LIN {X 0,Y 336.277,Z 972.972,A -85,B 0,C 180,E1 15001.794,E2 15001.794} C_VEL
LIN {X 0,Y 339.989,Z 961.244,A -85,B 0,C 180,E1 14998.442,E2 14998.442} C_VEL
LIN {X 0,Y 344.835,Z 946.848,A -85,B 0,C 180,E1 14994.971,E2 14994.971} C_VEL
LIN {X 0,Y 349.727,Z 932.706,A -85,B 0,C 180,E1 14992.08,E2 14992.08} C_VEL
LIN {X 0,Y 355.343,Z 916.384,A -85,B 0,C 180,E1 14989.256,E2 14989.256} C_VEL
LIN {X 0,Y 361.12,Z 899.297,A -85,B 0,C 180,E1 14986.734,E2 14986.734} C_VEL
LIN {X 0,Y 367.118,Z 880.482,A -85,B 0,C 180,E1 14984.422,E2 14984.422} C_VEL
LIN {X 0,Y 372.928,Z 861.29,A -85,B 0,C 180,E1 14982.427,E2 14982.427} C_VEL
LIN {X 0,Y 378.209,Z 842.054,A -85,B 0,C 180,E1 14980.766,E2 14980.766} C_VEL
LIN {X 0,Y 383.447,Z 821.063,A -85,B 0,C 180,E1 14979.255,E2 14979.255} C_VEL
LIN {X 0,Y 387.615,Z 801.784,A -85,B 0,C 180,E1 14978.127,E2 14978.127} C_VEL
LIN {X 0,Y 391.771,Z 779.558,A -85,B 0,C 180,E1 14977.076,E2 14977.076} C_VEL
LIN {X 0,Y 394.918,Z 758.505,A -85,B 0,C 180,E1 14976.32,E2 14976.32} C_VEL
LIN {X 0,Y 397.568,Z 734.492,A -85,B 0,C 180,E1 14975.675,E2 14975.675} C_VEL
LIN {X 0,Y 409.561,Z 529.671,A -85,B 0,C 180,E1 14971.616,E2 14971.616} C_VEL
LIN {X 0,Y 411.578,Z 493.902,A -85,B 0,C 180,E1 14970.88,E2 14970.88} C_VEL
LIN {X 0,Y 401.708,Z 478.08,A -85,B 0,C 180,E1 14968.102,E2 14968.102} C_VEL
LIN {X 0,Y 391.949,Z 463.545,A -85,B 0,C 180,E1 14965.053,E2 14965.053} C_VEL
LIN {X 0,Y 383.204,Z 451.285,A -85,B 0,C 180,E1 14961.988,E2 14961.988} C_VEL
LIN {X 0,Y 378.782,Z 445.758,A -85,B 0,C 180,E1 14960.31,E2 14960.31} C_VEL
LIN {X 0,Y 374.764,Z 440.732,A -85,B 0,C 180,E1 14958.672,E2 14958.672} C_VEL
LIN {X 0,Y 370.956,Z 435.952,A -85,B 0,C 180,E1 14957.004,E2 14957.004} C_VEL
LIN {X 0,Y 366.54,Z 430.926,A -85,B 0,C 180,E1 14954.938,E2 14954.938} C_VEL
LIN {X 0,Y 365.222,Z 429.224,A -85,B 0,C 180,E1 14954.263,E2 14954.263} C_VEL
LIN {X 0,Y 361.737,Z 425.607,A -85,B 0,C 180,E1 14952.45,E2 14952.45} C_VEL
LIN {X 0,Y 360.146,Z 423.216,A -85,B 0,C 180,E1 14951.508,E2 14951.508} C_VEL
LIN {X 0,Y 356.524,Z 419.861,A -85,B 0,C 180,E1 14949.361,E2 14949.361} C_VEL
LIN {X 0,Y 354.747,Z 416.927,A -85,B 0,C 180,E1 14948.101,E2 14948.101} C_VEL
LIN {X 0,Y 351.223,Z 414.2,A -85,B 0,C 180,E1 14945.636,E2 14945.636} C_VEL
LIN {X 0,Y 349.164,Z 410.557,A -85,B 0,C 180,E1 14943.776,E2 14943.776} C_VEL
LIN {X 0,Y 345.15,Z 407.759,A -85,B 0,C 180,E1 14939.999,E2 14939.999} C_VEL
LIN {X 0,Y 342.976,Z 403.947,A -85,B 0,C 180,E1 14936.991,E2 14936.991} C_VEL
LIN {X 0,Y 339.469,Z 401.855,A -85,B 0,C 180,E1 14929.992,E2 14929.992} C_VEL
LIN {X 0,Y 338.898,Z 401.219,A -85,B 0,C 180,E1 14924.715,E2 14924.715} C_VEL
LIN {X 0,Y 340.368,Z 402.502,A -85,B 0,C 180,E1 14918.605,E2 14918.605} C_VEL
LIN {X 0,Y 343.058,Z 404.045,A -85,B 0,C 180,E1 14914.075,E2 14914.075} C_VEL
LIN {X 0,Y 345.939,Z 408.538,A -85,B 0,C 180,E1 14910.38,E2 14910.38} C_VEL
LIN {X 0,Y 349.443,Z 410.923,A -85,B 0,C 180,E1 14907.213,E2 14907.213} C_VEL
LIN {X 0,Y 351.487,Z 414.448,A -85,B 0,C 180,E1 14905.423,E2 14905.423} C_VEL
LIN {X 0,Y 355.199,Z 417.46,A -85,B 0,C 180,E1 14902.857,E2 14902.857} C_VEL
LIN {X 0,Y 357.603,Z 421.145,A -85,B 0,C 180,E1 14901.221,E2 14901.221} C_VEL
LIN {X 0,Y 360.71,Z 423.864,A -85,B 0,C 180,E1 14899.446,E2 14899.446} C_VEL
LIN {X 0,Y 363.718,Z 427.939,A -85,B 0,C 180,E1 14897.768,E2 14897.768} C_VEL
LIN {X 0,Y 365.997,Z 430.022,A -85,B 0,C 180,E1 14896.637,E2 14896.637} C_VEL
LIN {X 0,Y 369.557,Z 434.555,A -85,B 0,C 180,E1 14894.914,E2 14894.914} C_VEL
LIN {X 0,Y 371.282,Z 436.471,A -85,B 0,C 180,E1 14894.136,E2 14894.136} C_VEL
LIN {X 0,Y 375.26,Z 441.146,A -85,B 0,C 180,E1 14892.433,E2 14892.433} C_VEL
LIN {X 0,Y 379.777,Z 446.735,A -85,B 0,C 180,E1 14890.627,E2 14890.627} C_VEL
LIN {X 0,Y 388.837,Z 458.356,A -85,B 0,C 180,E1 14887.355,E2 14887.355} C_VEL
LIN {X 0,Y 399.329,Z 472.434,A -85,B 0,C 180,E1 14884.026,E2 14884.026} C_VEL
LIN {X 0,Y 409.84,Z 487.637,A -85,B 0,C 180,E1 14881.057,E2 14881.057} C_VEL
LIN {X 0,Y 411.391,Z 490.242,A -85,B 0,C 180,E1 14880.637,E2 14880.637} C_VEL
LIN {X 0,Y 399.236,Z 697.815,A -85,B 0,C 180,E1 14876.553,E2 14876.553} C_VEL
LIN {X 0,Y 397.171,Z 724.706,A -85,B 0,C 180,E1 14875.953,E2 14875.953} C_VEL
LIN {X 0,Y 394.429,Z 747.684,A -85,B 0,C 180,E1 14875.24,E2 14875.24} C_VEL
LIN {X 0,Y 390.892,Z 769.549,A -85,B 0,C 180,E1 14874.313,E2 14874.313} C_VEL
LIN {X 0,Y 386.65,Z 791.514,A -85,B 0,C 180,E1 14873.139,E2 14873.139} C_VEL
LIN {X 0,Y 382.044,Z 811.473,A -85,B 0,C 180,E1 14871.81,E2 14871.81} C_VEL
LIN {X 0,Y 376.547,Z 832.601,A -85,B 0,C 180,E1 14870.107,E2 14870.107} C_VEL
LIN {X 0,Y 371.312,Z 850.638,A -85,B 0,C 180,E1 14868.358,E2 14868.358} C_VEL
LIN {X 0,Y 365.02,Z 870.569,A -85,B 0,C 180,E1 14866.055,E2 14866.055} C_VEL
LIN {X 0,Y 359.424,Z 887.312,A -85,B 0,C 180,E1 14863.754,E2 14863.754} C_VEL
LIN {X 0,Y 353.658,Z 903.672,A -85,B 0,C 180,E1 14861.079,E2 14861.079} C_VEL
LIN {X 0,Y 348.373,Z 918.498,A -85,B 0,C 180,E1 14858.245,E2 14858.245} C_VEL
LIN {X 0,Y 345.359,Z 926.835,A -85,B 0,C 180,E1 14856.41,E2 14856.41} C_VEL
LIN {X 0,Y 342.903,Z 931.412,A -85,B 0,C 180,E1 14855.448,E2 14855.448} C_VEL
LIN {X 0,Y 333.624,Z 942.542,A -85,B 0,C 180,E1 14853.077,E2 14853.077} C_VEL
LIN {X 0,Y 331.307,Z 946.444,A -85,B 0,C 180,E1 14851.991,E2 14851.991} C_VEL
LIN {X 0,Y 327.771,Z 956.623,A -85,B 0,C 180,E1 14848.596,E2 14848.596} C_VEL
LIN {X 0,Y 324.573,Z 966.727,A -85,B 0,C 180,E1 14844.515,E2 14844.515} C_VEL
LIN {X 0,Y 322.438,Z 974.749,A -85,B 0,C 180,E1 14840.535,E2 14840.535} C_VEL
LIN {X 0,Y 321.058,Z 981.036,A -85,B 0,C 180,E1 14836.488,E2 14836.488} C_VEL
LIN {X 0,Y 320.354,Z 985.736,A -85,B 0,C 180,E1 14832.56,E2 14832.56} C_VEL
LIN {X 0,Y 320.061,Z 988.751,A -85,B 0,C 180,E1 14828.749,E2 14828.749} C_VEL
LIN {X 0,Y 319.978,Z 990.434,A -85,B 0,C 180,E1 14825.241,E2 14825.241} C_VEL
LIN {X 0,Y 319.967,Z 990.942,A -85,B 0,C 180,E1 14821.229,E2 14821.229} C_VEL
LIN {X 0,Y 319.978,Z 990.216,A -85,B 0,C 180,E1 14817.868,E2 14817.868} C_VEL
LIN {X 0,Y 320.126,Z 988.191,A -85,B 0,C 180,E1 14813.994,E2 14813.994} C_VEL
LIN {X 0,Y 320.55,Z 984.512,A -85,B 0,C 180,E1 14810.012,E2 14810.012} C_VEL
LIN {X 0,Y 321.476,Z 979.566,A -85,B 0,C 180,E1 14806.081,E2 14806.081} C_VEL
LIN {X 0,Y 323.018,Z 973.025,A -85,B 0,C 180,E1 14802.199,E2 14802.199} C_VEL
LIN {X 0,Y 325.366,Z 965.15,A -85,B 0,C 180,E1 14798.372,E2 14798.372} C_VEL
LIN {X 0,Y 328.589,Z 955.458,A -85,B 0,C 180,E1 14794.59,E2 14794.59} C_VEL
LIN {X 0,Y 332.897,Z 943.804,A -85,B 0,C 180,E1 14790.789,E2 14790.789} C_VEL
LIN {X 0,Y 337.523,Z 931.777,A -85,B 0,C 180,E1 14787.525,E2 14787.525} C_VEL
LIN {X 0,Y 343.347,Z 917.072,A -85,B 0,C 180,E1 14784.169,E2 14784.169} C_VEL
LIN {X 0,Y 349.136,Z 902.312,A -85,B 0,C 180,E1 14781.329,E2 14781.329} C_VEL
LIN {X 0,Y 355.55,Z 885.443,A -85,B 0,C 180,E1 14778.605,E2 14778.605} C_VEL
LIN {X 0,Y 362.016,Z 867.798,A -85,B 0,C 180,E1 14776.198,E2 14776.198} C_VEL
LIN {X 0,Y 368.118,Z 849.666,A -85,B 0,C 180,E1 14774.139,E2 14774.139} C_VEL
LIN {X 0,Y 374.231,Z 830.086,A -85,B 0,C 180,E1 14772.264,E2 14772.264} C_VEL
LIN {X 0,Y 379.729,Z 810.272,A -85,B 0,C 180,E1 14770.699,E2 14770.699} C_VEL
LIN {X 0,Y 385.279,Z 787.324,A -85,B 0,C 180,E1 14769.222,E2 14769.222} C_VEL
LIN {X 0,Y 389.546,Z 766.561,A -85,B 0,C 180,E1 14768.153,E2 14768.153} C_VEL
LIN {X 0,Y 393.289,Z 743.628,A -85,B 0,C 180,E1 14767.242,E2 14767.242} C_VEL
LIN {X 0,Y 396.188,Z 720.474,A -85,B 0,C 180,E1 14766.565,E2 14766.565} C_VEL
LIN {X 0,Y 403.462,Z 618.117,A -85,B 0,C 180,E1 14764.456,E2 14764.456} C_VEL
LIN {X 0,Y 412.474,Z 496.118,A -85,B 0,C 180,E1 14761.945,E2 14761.945} C_VEL
LIN {X 0,Y 406.567,Z 486.319,A -85,B 0,C 180,E1 14759.578,E2 14759.578} C_VEL
LIN {X 0,Y 401.968,Z 478.937,A -85,B 0,C 180,E1 14757.363,E2 14757.363} C_VEL
LIN {X 0,Y 399.286,Z 474.781,A -85,B 0,C 180,E1 14755.836,E2 14755.836} C_VEL
LIN {X 0,Y 396.693,Z 470.696,A -85,B 0,C 180,E1 14754.069,E2 14754.069} C_VEL
LIN {X 0,Y 394.074,Z 466.488,A -85,B 0,C 180,E1 14751.685,E2 14751.685} C_VEL
LIN {X 0,Y 393.166,Z 465.528,A -85,B 0,C 180,E1 14750.634,E2 14750.634} C_VEL
LIN {X 0,Y 391.561,Z 463.129,A -85,B 0,C 180,E1 14746.638,E2 14746.638} C_VEL
LIN {X 0,Y 391.761,Z 463.738,A -85,B 0,C 180,E1 14744.456,E2 14744.456} C_VEL
LIN {X 0,Y 394.02,Z 466.346,A -85,B 0,C 180,E1 14740.816,E2 14740.816} C_VEL
LIN {X 0,Y 396.488,Z 470.513,A -85,B 0,C 180,E1 14738.525,E2 14738.525} C_VEL
LIN {X 0,Y 397.564,Z 472.154,A -85,B 0,C 180,E1 14737.729,E2 14737.729} C_VEL
LIN {X 0,Y 400.699,Z 477.067,A -85,B 0,C 180,E1 14735.766,E2 14735.766} C_VEL
LIN {X 0,Y 405.039,Z 484.946,A -85,B 0,C 180,E1 14733.501,E2 14733.501} C_VEL
LIN {X 0,Y 410.015,Z 494.373,A -85,B 0,C 180,E1 14731.329,E2 14731.329} C_VEL
LIN {X 0,Y 412.455,Z 499.516,A -85,B 0,C 180,E1 14730.365,E2 14730.365} C_VEL
LIN {X 0,Y 398.746,Z 689.757,A -85,B 0,C 180,E1 14726.482,E2 14726.482} C_VEL
LIN {X 0,Y 395.345,Z 736.083,A -85,B 0,C 180,E1 14725.504,E2 14725.504} C_VEL
LIN {X 0,Y 392.335,Z 758.929,A -85,B 0,C 180,E1 14724.859,E2 14724.859} C_VEL
LIN {X 0,Y 388.399,Z 781.737,A -85,B 0,C 180,E1 14724,E2 14724} C_VEL
LIN {X 0,Y 384.215,Z 801.576,A -85,B 0,C 180,E1 14723.031,E2 14723.031} C_VEL
LIN {X 0,Y 378.701,Z 824.282,A -85,B 0,C 180,E1 14721.647,E2 14721.647} C_VEL
LIN {X 0,Y 373.434,Z 843.326,A -85,B 0,C 180,E1 14720.218,E2 14720.218} C_VEL
LIN {X 0,Y 366.723,Z 865.269,A -85,B 0,C 180,E1 14718.223,E2 14718.223} C_VEL
LIN {X 0,Y 360.501,Z 884.173,A -85,B 0,C 180,E1 14716.151,E2 14716.151} C_VEL
LIN {X 0,Y 354.121,Z 902.261,A -85,B 0,C 180,E1 14713.774,E2 14713.774} C_VEL
LIN {X 0,Y 347.818,Z 919.74,A -85,B 0,C 180,E1 14711.066,E2 14711.066} C_VEL
LIN {X 0,Y 341.862,Z 935.706,A -85,B 0,C 180,E1 14708.111,E2 14708.111} C_VEL
LIN {X 0,Y 336.071,Z 951.541,A -85,B 0,C 180,E1 14704.633,E2 14704.633} C_VEL
LIN {X 0,Y 331.503,Z 964.51,A -85,B 0,C 180,E1 14701.255,E2 14701.255} C_VEL
LIN {X 0,Y 327.475,Z 976.677,A -85,B 0,C 180,E1 14697.459,E2 14697.459} C_VEL
LIN {X 0,Y 324.466,Z 987.037,A -85,B 0,C 180,E1 14693.621,E2 14693.621} C_VEL
LIN {X 0,Y 322.36,Z 995.464,A -85,B 0,C 180,E1 14689.765,E2 14689.765} C_VEL
LIN {X 0,Y 320.975,Z 1002.68,A -85,B 0,C 180,E1 14685.729,E2 14685.729} C_VEL
LIN {X 0,Y 320.293,Z 1007.657,A -85,B 0,C 180,E1 14682.078,E2 14682.078} C_VEL
LIN {X 0,Y 320.024,Z 1011.558,A -85,B 0,C 180,E1 14678.268,E2 14678.268} C_VEL
LIN {X 0,Y 319.947,Z 1013.919,A -85,B 0,C 180,E1 14674.486,E2 14674.486} C_VEL
LIN {X 0,Y 319.954,Z 1014.85,A -85,B 0,C 180,E1 14671.259,E2 14671.259} C_VEL
LIN {X 0,Y 319.957,Z 1014.756,A -85,B 0,C 180,E1 14667.856,E2 14667.856} C_VEL
LIN {X 0,Y 319.961,Z 1013.15,A -85,B 0,C 180,E1 14663.907,E2 14663.907} C_VEL
LIN {X 0,Y 320.07,Z 1010.516,A -85,B 0,C 180,E1 14660.476,E2 14660.476} C_VEL
LIN {X 0,Y 320.522,Z 1006.051,A -85,B 0,C 180,E1 14656.476,E2 14656.476} C_VEL
LIN {X 0,Y 321.458,Z 1000.137,A -85,B 0,C 180,E1 14652.633,E2 14652.633} C_VEL
LIN {X 0,Y 323.16,Z 992.342,A -85,B 0,C 180,E1 14648.593,E2 14648.593} C_VEL
LIN {X 0,Y 325.507,Z 983.552,A -85,B 0,C 180,E1 14644.926,E2 14644.926} C_VEL
LIN {X 0,Y 328.905,Z 972.591,A -85,B 0,C 180,E1 14641.103,E2 14641.103} C_VEL
LIN {X 0,Y 332.857,Z 960.835,A -85,B 0,C 180,E1 14637.685,E2 14637.685} C_VEL
LIN {X 0,Y 337.971,Z 946.399,A -85,B 0,C 180,E1 14634.151,E2 14634.151} C_VEL
LIN {X 0,Y 343.469,Z 931.373,A -85,B 0,C 180,E1 14631.048,E2 14631.048} C_VEL
LIN {X 0,Y 349.382,Z 914.816,A -85,B 0,C 180,E1 14628.188,E2 14628.188} C_VEL
LIN {X 0,Y 355.647,Z 896.985,A -85,B 0,C 180,E1 14625.579,E2 14625.579} C_VEL
LIN {X 0,Y 361.661,Z 878.859,A -85,B 0,C 180,E1 14623.366,E2 14623.366} C_VEL
LIN {X 0,Y 368.154,Z 857.85,A -85,B 0,C 180,E1 14621.22,E2 14621.22} C_VEL
LIN {X 0,Y 373.6,Z 838.56,A -85,B 0,C 180,E1 14619.587,E2 14619.587} C_VEL
LIN {X 0,Y 378.791,Z 817.787,A -85,B 0,C 180,E1 14618.141,E2 14618.141} C_VEL
LIN {X 0,Y 383.417,Z 796.805,A -85,B 0,C 180,E1 14616.949,E2 14616.949} C_VEL
LIN {X 0,Y 387.543,Z 774.028,A -85,B 0,C 180,E1 14615.94,E2 14615.94} C_VEL
LIN {X 0,Y 390.938,Z 751.015,A -85,B 0,C 180,E1 14615.171,E2 14615.171} C_VEL
LIN {X 0,Y 393.173,Z 727.848,A -85,B 0,C 180,E1 14614.609,E2 14614.609} C_VEL
LIN {X 0,Y 405.857,Z 518.019,A -85,B 0,C 180,E1 14610.446,E2 14610.446} C_VEL
LIN {X 0,Y 407.024,Z 498.197,A -85,B 0,C 180,E1 14610.033,E2 14610.033} C_VEL
LIN {X 0,Y 398.344,Z 484.149,A -85,B 0,C 180,E1 14607.506,E2 14607.506} C_VEL
LIN {X 0,Y 389.062,Z 470.099,A -85,B 0,C 180,E1 14604.521,E2 14604.521} C_VEL
LIN {X 0,Y 380.64,Z 458.182,A -85,B 0,C 180,E1 14601.495,E2 14601.495} C_VEL
LIN {X 0,Y 376.458,Z 452.884,A -85,B 0,C 180,E1 14599.874,E2 14599.874} C_VEL
LIN {X 0,Y 372.491,Z 447.9,A -85,B 0,C 180,E1 14598.222,E2 14598.222} C_VEL
LIN {X 0,Y 368.096,Z 442.463,A -85,B 0,C 180,E1 14596.246,E2 14596.246} C_VEL
LIN {X 0,Y 364.285,Z 437.786,A -85,B 0,C 180,E1 14594.382,E2 14594.382} C_VEL
LIN {X 0,Y 359.675,Z 432.659,A -85,B 0,C 180,E1 14591.93,E2 14591.93} C_VEL
LIN {X 0,Y 358.575,Z 430.922,A -85,B 0,C 180,E1 14591.255,E2 14591.255} C_VEL
LIN {X 0,Y 354.951,Z 427.511,A -85,B 0,C 180,E1 14589.075,E2 14589.075} C_VEL
LIN {X 0,Y 353.175,Z 424.649,A -85,B 0,C 180,E1 14587.801,E2 14587.801} C_VEL
LIN {X 0,Y 349.731,Z 421.837,A -85,B 0,C 180,E1 14585.331,E2 14585.331} C_VEL
LIN {X 0,Y 347.677,Z 418.278,A -85,B 0,C 180,E1 14583.462,E2 14583.462} C_VEL
LIN {X 0,Y 343.903,Z 415.6,A -85,B 0,C 180,E1 14579.833,E2 14579.833} C_VEL
LIN {X 0,Y 341.756,Z 411.788,A -85,B 0,C 180,E1 14576.813,E2 14576.813} C_VEL
LIN {X 0,Y 338.282,Z 409.684,A -85,B 0,C 180,E1 14569.612,E2 14569.612} C_VEL
LIN {X 0,Y 337.832,Z 409.17,A -85,B 0,C 180,E1 14564.551,E2 14564.551} C_VEL
LIN {X 0,Y 339.384,Z 410.502,A -85,B 0,C 180,E1 14558.391,E2 14558.391} C_VEL
LIN {X 0,Y 341.903,Z 411.948,A -85,B 0,C 180,E1 14554.167,E2 14554.167} C_VEL
LIN {X 0,Y 344.433,Z 416.115,A -85,B 0,C 180,E1 14550.81,E2 14550.81} C_VEL
LIN {X 0,Y 347.994,Z 418.665,A -85,B 0,C 180,E1 14547.5,E2 14547.5} C_VEL
LIN {X 0,Y 350.185,Z 422.312,A -85,B 0,C 180,E1 14545.574,E2 14545.574} C_VEL
LIN {X 0,Y 353.601,Z 425.138,A -85,B 0,C 180,E1 14543.168,E2 14543.168} C_VEL
LIN {X 0,Y 356.254,Z 429.032,A -85,B 0,C 180,E1 14541.356,E2 14541.356} C_VEL
LIN {X 0,Y 359.022,Z 431.532,A -85,B 0,C 180,E1 14539.75,E2 14539.75} C_VEL
LIN {X 0,Y 362.254,Z 435.766,A -85,B 0,C 180,E1 14537.932,E2 14537.932} C_VEL
LIN {X 0,Y 364.229,Z 437.693,A -85,B 0,C 180,E1 14536.932,E2 14536.932} C_VEL
LIN {X 0,Y 367.883,Z 442.241,A -85,B 0,C 180,E1 14535.146,E2 14535.146} C_VEL
LIN {X 0,Y 369.66,Z 444.453,A -85,B 0,C 180,E1 14534.321,E2 14534.321} C_VEL
LIN {X 0,Y 374.201,Z 450.014,A -85,B 0,C 180,E1 14532.358,E2 14532.358} C_VEL
LIN {X 0,Y 378.931,Z 455.989,A -85,B 0,C 180,E1 14530.466,E2 14530.466} C_VEL
LIN {X 0,Y 384.137,Z 462.62,A -85,B 0,C 180,E1 14528.54,E2 14528.54} C_VEL
LIN {X 0,Y 391.773,Z 472.822,A -85,B 0,C 180,E1 14525.954,E2 14525.954} C_VEL
LIN {X 0,Y 399.937,Z 484.207,A -85,B 0,C 180,E1 14523.447,E2 14523.447} C_VEL
LIN {X 0,Y 406.789,Z 494.512,A -85,B 0,C 180,E1 14521.499,E2 14521.499} C_VEL
LIN {X 0,Y 394.119,Z 703.148,A -85,B 0,C 180,E1 14517.375,E2 14517.375} C_VEL
LIN {X 0,Y 392.075,Z 726.879,A -85,B 0,C 180,E1 14516.82,E2 14516.82} C_VEL
LIN {X 0,Y 389.066,Z 750.34,A -85,B 0,C 180,E1 14516.063,E2 14516.063} C_VEL
LIN {X 0,Y 385.671,Z 770.502,A -85,B 0,C 180,E1 14515.197,E2 14515.197} C_VEL
LIN {X 0,Y 381.161,Z 792.857,A -85,B 0,C 180,E1 14513.985,E2 14513.985} C_VEL
LIN {X 0,Y 376.645,Z 811.811,A -85,B 0,C 180,E1 14512.715,E2 14512.715} C_VEL
LIN {X 0,Y 370.955,Z 832.98,A -85,B 0,C 180,E1 14511.001,E2 14511.001} C_VEL
LIN {X 0,Y 365.525,Z 851.03,A -85,B 0,C 180,E1 14509.24,E2 14509.24} C_VEL
LIN {X 0,Y 358.981,Z 870.958,A -85,B 0,C 180,E1 14506.916,E2 14506.916} C_VEL
LIN {X 0,Y 352.971,Z 888.244,A -85,B 0,C 180,E1 14504.513,E2 14504.513} C_VEL
LIN {X 0,Y 346.968,Z 904.539,A -85,B 0,C 180,E1 14501.801,E2 14501.801} C_VEL
LIN {X 0,Y 341.454,Z 919.307,A -85,B 0,C 180,E1 14498.923,E2 14498.923} C_VEL
LIN {X 0,Y 336.346,Z 932.716,A -85,B 0,C 180,E1 14495.795,E2 14495.795} C_VEL
LIN {X 0,Y 331.601,Z 945.647,A -85,B 0,C 180,E1 14492.241,E2 14492.241} C_VEL
LIN {X 0,Y 331.307,Z 946.444,A -85,B 0,C 180,E1 14491.991,E2 14491.991} C_VEL
LIN {X 0,Y 329.061,Z 950.294,A -85,B 0,C 180,E1 14490.878,E2 14490.878} C_VEL
LIN {X 0,Y 319.962,Z 960.084,A -85,B 0,C 180,E1 14487.96,E2 14487.96} C_VEL
LIN {X 0,Y 318.317,Z 962.79,A -85,B 0,C 180,E1 14486.915,E2 14486.915} C_VEL
LIN {X 0,Y 315.495,Z 971.833,A -85,B 0,C 180,E1 14482.712,E2 14482.712} C_VEL
LIN {X 0,Y 313.818,Z 978.282,A -85,B 0,C 180,E1 14478.974,E2 14478.974} C_VEL
LIN {X 0,Y 312.664,Z 984.089,A -85,B 0,C 180,E1 14474.603,E2 14474.603} C_VEL
LIN {X 0,Y 312.198,Z 987.465,A -85,B 0,C 180,E1 14471.122,E2 14471.122} C_VEL
LIN {X 0,Y 312.007,Z 990.048,A -85,B 0,C 180,E1 14467.18,E2 14467.18} C_VEL
LIN {X 0,Y 311.956,Z 991.133,A -85,B 0,C 180,E1 14463.411,E2 14463.411} C_VEL
LIN {X 0,Y 311.954,Z 991.112,A -85,B 0,C 180,E1 14459.995,E2 14459.995} C_VEL
LIN {X 0,Y 312.018,Z 989.858,A -85,B 0,C 180,E1 14456.096,E2 14456.096} C_VEL
LIN {X 0,Y 312.24,Z 987.471,A -85,B 0,C 180,E1 14452.519,E2 14452.519} C_VEL
LIN {X 0,Y 312.812,Z 983.758,A -85,B 0,C 180,E1 14448.691,E2 14448.691} C_VEL
LIN {X 0,Y 314.044,Z 978.025,A -85,B 0,C 180,E1 14444.463,E2 14444.463} C_VEL
LIN {X 0,Y 316.104,Z 970.865,A -85,B 0,C 180,E1 14440.327,E2 14440.327} C_VEL
LIN {X 0,Y 319.007,Z 962.036,A -85,B 0,C 180,E1 14436.327,E2 14436.327} C_VEL
LIN {X 0,Y 323.03,Z 951.337,A -85,B 0,C 180,E1 14432.321,E2 14432.321} C_VEL
LIN {X 0,Y 327.537,Z 940.002,A -85,B 0,C 180,E1 14428.816,E2 14428.816} C_VEL
LIN {X 0,Y 333.312,Z 926.039,A -85,B 0,C 180,E1 14425.213,E2 14425.213} C_VEL
LIN {X 0,Y 339.437,Z 911.427,A -85,B 0,C 180,E1 14422.051,E2 14422.051} C_VEL
LIN {X 0,Y 345.741,Z 895.864,A -85,B 0,C 180,E1 14419.25,E2 14419.25} C_VEL
LIN {X 0,Y 352.634,Z 878.365,A -85,B 0,C 180,E1 14416.582,E2 14416.582} C_VEL
LIN {X 0,Y 359.144,Z 860.624,A -85,B 0,C 180,E1 14414.332,E2 14414.332} C_VEL
LIN {X 0,Y 366.174,Z 840,A -85,B 0,C 180,E1 14412.155,E2 14412.155} C_VEL
LIN {X 0,Y 372.151,Z 820.633,A -85,B 0,C 180,E1 14410.462,E2 14410.462} C_VEL
LIN {X 0,Y 377.731,Z 800.016,A -85,B 0,C 180,E1 14408.985,E2 14408.985} C_VEL
LIN {X 0,Y 382.61,Z 779.456,A -85,B 0,C 180,E1 14407.777,E2 14407.777} C_VEL
LIN {X 0,Y 386.801,Z 757.712,A -85,B 0,C 180,E1 14406.771,E2 14406.771} C_VEL
LIN {X 0,Y 390.304,Z 735.408,A -85,B 0,C 180,E1 14405.971,E2 14405.971} C_VEL
LIN {X 0,Y 392.742,Z 712.745,A -85,B 0,C 180,E1 14405.391,E2 14405.391} C_VEL
LIN {X 0,Y 408.409,Z 506.179,A -85,B 0,C 180,E1 14401.154,E2 14401.154} C_VEL
LIN {X 0,Y 408.741,Z 500.898,A -85,B 0,C 180,E1 14401.017,E2 14401.017} C_VEL
LIN {X 0,Y 403.256,Z 491.362,A -85,B 0,C 180,E1 14398.615,E2 14398.615} C_VEL
LIN {X 0,Y 398.357,Z 483.284,A -85,B 0,C 180,E1 14395.971,E2 14395.971} C_VEL
LIN {X 0,Y 395.153,Z 478.287,A -85,B 0,C 180,E1 14393.754,E2 14393.754} C_VEL
LIN {X 0,Y 392.674,Z 474.041,A -85,B 0,C 180,E1 14391.36,E2 14391.36} C_VEL
LIN {X 0,Y 390.494,Z 471.172,A -85,B 0,C 180,E1 14386.979,E2 14386.979} C_VEL
LIN {X 0,Y 390.535,Z 471.273,A -85,B 0,C 180,E1 14385.166,E2 14385.166} C_VEL
LIN {X 0,Y 392.754,Z 474.252,A -85,B 0,C 180,E1 14380.983,E2 14380.983} C_VEL
LIN {X 0,Y 395.22,Z 478.394,A -85,B 0,C 180,E1 14378.636,E2 14378.636} C_VEL
LIN {X 0,Y 398.844,Z 484.355,A -85,B 0,C 180,E1 14376.157,E2 14376.157} C_VEL
LIN {X 0,Y 403.442,Z 492.993,A -85,B 0,C 180,E1 14373.666,E2 14373.666} C_VEL
LIN {X 0,Y 408.76,Z 503.676,A -85,B 0,C 180,E1 14371.298,E2 14371.298} C_VEL
LIN {X 0,Y 394.509,Z 692.288,A -85,B 0,C 180,E1 14367.431,E2 14367.431} C_VEL
LIN {X 0,Y 391.129,Z 736.031,A -85,B 0,C 180,E1 14366.501,E2 14366.501} C_VEL
LIN {X 0,Y 387.99,Z 758.915,A -85,B 0,C 180,E1 14365.852,E2 14365.852} C_VEL
LIN {X 0,Y 383.757,Z 782.304,A -85,B 0,C 180,E1 14364.966,E2 14364.966} C_VEL
LIN {X 0,Y 379.442,Z 801.994,A -85,B 0,C 180,E1 14364,E2 14364} C_VEL
LIN {X 0,Y 373.735,Z 824.467,A -85,B 0,C 180,E1 14362.619,E2 14362.619} C_VEL
LIN {X 0,Y 368.279,Z 843.4,A -85,B 0,C 180,E1 14361.191,E2 14361.191} C_VEL
LIN {X 0,Y 361.533,Z 864.591,A -85,B 0,C 180,E1 14359.257,E2 14359.257} C_VEL
LIN {X 0,Y 355.068,Z 883.393,A -85,B 0,C 180,E1 14357.19,E2 14357.19} C_VEL
LIN {X 0,Y 348.379,Z 901.522,A -85,B 0,C 180,E1 14354.801,E2 14354.801} C_VEL
LIN {X 0,Y 341.762,Z 919.046,A -85,B 0,C 180,E1 14352.069,E2 14352.069} C_VEL
LIN {X 0,Y 335.651,Z 934.584,A -85,B 0,C 180,E1 14349.167,E2 14349.167} C_VEL
LIN {X 0,Y 329.765,Z 949.824,A -85,B 0,C 180,E1 14345.821,E2 14345.821} C_VEL
LIN {X 0,Y 325.024,Z 962.319,A -85,B 0,C 180,E1 14342.554,E2 14342.554} C_VEL
LIN {X 0,Y 320.431,Z 975.307,A -85,B 0,C 180,E1 14338.522,E2 14338.522} C_VEL
LIN {X 0,Y 317.245,Z 985.323,A -85,B 0,C 180,E1 14334.787,E2 14334.787} C_VEL
LIN {X 0,Y 314.754,Z 994.417,A -85,B 0,C 180,E1 14330.652,E2 14330.652} C_VEL
LIN {X 0,Y 313.242,Z 1001.486,A -85,B 0,C 180,E1 14326.7,E2 14326.7} C_VEL
LIN {X 0,Y 312.366,Z 1007.132,A -85,B 0,C 180,E1 14322.577,E2 14322.577} C_VEL
LIN {X 0,Y 312.043,Z 1010.919,A -85,B 0,C 180,E1 14318.853,E2 14318.853} C_VEL
LIN {X 0,Y 311.95,Z 1013.545,A -85,B 0,C 180,E1 14314.786,E2 14314.786} C_VEL
LIN {X 0,Y 311.96,Z 1014.55,A -85,B 0,C 180,E1 14311.291,E2 14311.291} C_VEL
LIN {X 0,Y 311.961,Z 1014.456,A -85,B 0,C 180,E1 14307.801,E2 14307.801} C_VEL
LIN {X 0,Y 311.968,Z 1012.846,A -85,B 0,C 180,E1 14303.75,E2 14303.75} C_VEL
LIN {X 0,Y 312.079,Z 1010.206,A -85,B 0,C 180,E1 14300.23,E2 14300.23} C_VEL
LIN {X 0,Y 312.579,Z 1005.727,A -85,B 0,C 180,E1 14296.125,E2 14296.125} C_VEL
LIN {X 0,Y 313.531,Z 1000.115,A -85,B 0,C 180,E1 14292.371,E2 14292.371} C_VEL
LIN {X 0,Y 315.297,Z 992.563,A -85,B 0,C 180,E1 14288.301,E2 14288.301} C_VEL
LIN {X 0,Y 317.808,Z 983.659,A -85,B 0,C 180,E1 14284.475,E2 14284.475} C_VEL
LIN {X 0,Y 321.388,Z 972.777,A -85,B 0,C 180,E1 14280.565,E2 14280.565} C_VEL
LIN {X 0,Y 325.536,Z 961.068,A -85,B 0,C 180,E1 14277.076,E2 14277.076} C_VEL
LIN {X 0,Y 330.892,Z 946.734,A -85,B 0,C 180,E1 14273.476,E2 14273.476} C_VEL
LIN {X 0,Y 336.28,Z 932.608,A -85,B 0,C 180,E1 14270.493,E2 14270.493} C_VEL
LIN {X 0,Y 342.591,Z 915.823,A -85,B 0,C 180,E1 14267.505,E2 14267.505} C_VEL
LIN {X 0,Y 349.083,Z 898.232,A -85,B 0,C 180,E1 14264.864,E2 14264.864} C_VEL
LIN {X 0,Y 355.389,Z 879.939,A -85,B 0,C 180,E1 14262.59,E2 14262.59} C_VEL
LIN {X 0,Y 361.745,Z 860.371,A -85,B 0,C 180,E1 14260.537,E2 14260.537} C_VEL
LIN {X 0,Y 367.33,Z 841.384,A -85,B 0,C 180,E1 14258.889,E2 14258.889} C_VEL
LIN {X 0,Y 372.942,Z 820.249,A -85,B 0,C 180,E1 14257.363,E2 14257.363} C_VEL
LIN {X 0,Y 377.68,Z 799.637,A -85,B 0,C 180,E1 14256.164,E2 14256.164} C_VEL
LIN {X 0,Y 382.315,Z 775.529,A -85,B 0,C 180,E1 14255.06,E2 14255.06} C_VEL
LIN {X 0,Y 385.786,Z 753.141,A -85,B 0,C 180,E1 14254.293,E2 14254.293} C_VEL
LIN {X 0,Y 388.243,Z 729.49,A -85,B 0,C 180,E1 14253.703,E2 14253.703} C_VEL
LIN {X 0,Y 401.452,Z 519.877,A -85,B 0,C 180,E1 14249.52,E2 14249.52} C_VEL
LIN {X 0,Y 402.471,Z 502.289,A -85,B 0,C 180,E1 14249.138,E2 14249.138} C_VEL
LIN {X 0,Y 393.875,Z 488.39,A -85,B 0,C 180,E1 14246.537,E2 14246.537} C_VEL
LIN {X 0,Y 384.83,Z 474.576,A -85,B 0,C 180,E1 14243.504,E2 14243.504} C_VEL
LIN {X 0,Y 377.162,Z 463.91,A -85,B 0,C 180,E1 14240.645,E2 14240.645} C_VEL
LIN {X 0,Y 373.982,Z 459.803,A -85,B 0,C 180,E1 14239.36,E2 14239.36} C_VEL
LIN {X 0,Y 370.233,Z 455.051,A -85,B 0,C 180,E1 14237.768,E2 14237.768} C_VEL
LIN {X 0,Y 365.902,Z 449.666,A -85,B 0,C 180,E1 14235.776,E2 14235.776} C_VEL
LIN {X 0,Y 361.584,Z 444.303,A -85,B 0,C 180,E1 14233.594,E2 14233.594} C_VEL
LIN {X 0,Y 357.959,Z 440.217,A -85,B 0,C 180,E1 14231.601,E2 14231.601} C_VEL
LIN {X 0,Y 356.678,Z 438.409,A -85,B 0,C 180,E1 14230.825,E2 14230.825} C_VEL
LIN {X 0,Y 353.048,Z 434.669,A -85,B 0,C 180,E1 14228.55,E2 14228.55} C_VEL
LIN {X 0,Y 351.629,Z 432.379,A -85,B 0,C 180,E1 14227.515,E2 14227.515} C_VEL
LIN {X 0,Y 348.143,Z 429.343,A -85,B 0,C 180,E1 14224.942,E2 14224.942} C_VEL
LIN {X 0,Y 346.393,Z 426.132,A -85,B 0,C 180,E1 14223.309,E2 14223.309} C_VEL
LIN {X 0,Y 342.659,Z 423.44,A -85,B 0,C 180,E1 14219.665,E2 14219.665} C_VEL
LIN {X 0,Y 340.51,Z 419.603,A -85,B 0,C 180,E1 14216.591,E2 14216.591} C_VEL
LIN {X 0,Y 337.11,Z 417.511,A -85,B 0,C 180,E1 14209.23,E2 14209.23} C_VEL
LIN {X 0,Y 336.772,Z 417.14,A -85,B 0,C 180,E1 14204.325,E2 14204.325} C_VEL
LIN {X 0,Y 338.417,Z 418.521,A -85,B 0,C 180,E1 14198.144,E2 14198.144} C_VEL
LIN {X 0,Y 340.758,Z 419.864,A -85,B 0,C 180,E1 14194.248,E2 14194.248} C_VEL
LIN {X 0,Y 343.102,Z 423.865,A -85,B 0,C 180,E1 14191.068,E2 14191.068} C_VEL
LIN {X 0,Y 346.596,Z 426.507,A -85,B 0,C 180,E1 14187.744,E2 14187.744} C_VEL
LIN {X 0,Y 348.886,Z 430.171,A -85,B 0,C 180,E1 14185.726,E2 14185.726} C_VEL
LIN {X 0,Y 352.053,Z 432.898,A -85,B 0,C 180,E1 14183.443,E2 14183.443} C_VEL
LIN {X 0,Y 354.903,Z 436.913,A -85,B 0,C 180,E1 14181.492,E2 14181.492} C_VEL
LIN {X 0,Y 357.299,Z 439.1,A -85,B 0,C 180,E1 14180.087,E2 14180.087} C_VEL
LIN {X 0,Y 360.633,Z 443.445,A -85,B 0,C 180,E1 14178.18,E2 14178.18} C_VEL
LIN {X 0,Y 362.497,Z 445.382,A -85,B 0,C 180,E1 14177.217,E2 14177.217} C_VEL
LIN {X 0,Y 366.482,Z 450.166,A -85,B 0,C 180,E1 14175.259,E2 14175.259} C_VEL
LIN {X 0,Y 372.349,Z 457.705,A -85,B 0,C 180,E1 14172.627,E2 14172.627} C_VEL
LIN {X 0,Y 376.708,Z 463.264,A -85,B 0,C 180,E1 14170.847,E2 14170.847} C_VEL
LIN {X 0,Y 383.445,Z 471.868,A -85,B 0,C 180,E1 14168.344,E2 14168.344} C_VEL
LIN {X 0,Y 393.797,Z 486.198,A -85,B 0,C 180,E1 14164.904,E2 14164.904} C_VEL
LIN {X 0,Y 402.259,Z 498.806,A -85,B 0,C 180,E1 14162.379,E2 14162.379} C_VEL
LIN {X 0,Y 388.995,Z 708.411,A -85,B 0,C 180,E1 14158.209,E2 14158.209} C_VEL
LIN {X 0,Y 386.868,Z 730.798,A -85,B 0,C 180,E1 14157.66,E2 14157.66} C_VEL
LIN {X 0,Y 383.631,Z 753.87,A -85,B 0,C 180,E1 14156.873,E2 14156.873} C_VEL
LIN {X 0,Y 380.048,Z 774.163,A -85,B 0,C 180,E1 14155.973,E2 14155.973} C_VEL
LIN {X 0,Y 375.507,Z 795.247,A -85,B 0,C 180,E1 14154.789,E2 14154.789} C_VEL
LIN {X 0,Y 370.63,Z 814.907,A -85,B 0,C 180,E1 14153.442,E2 14153.442} C_VEL
LIN {X 0,Y 364.748,Z 835.573,A -85,B 0,C 180,E1 14151.714,E2 14151.714} C_VEL
LIN {X 0,Y 358.736,Z 854.816,A -85,B 0,C 180,E1 14149.788,E2 14149.788} C_VEL
LIN {X 0,Y 352.432,Z 873.013,A -85,B 0,C 180,E1 14147.588,E2 14147.588} C_VEL
LIN {X 0,Y 346.016,Z 890.608,A -85,B 0,C 180,E1 14145.068,E2 14145.068} C_VEL
LIN {X 0,Y 339.992,Z 906.24,A -85,B 0,C 180,E1 14142.391,E2 14142.391} C_VEL
LIN {X 0,Y 333.667,Z 922.274,A -85,B 0,C 180,E1 14139.133,E2 14139.133} C_VEL
LIN {X 0,Y 328.482,Z 935.458,A -85,B 0,C 180,E1 14135.935,E2 14135.935} C_VEL
LIN {X 0,Y 323.626,Z 947.96,A -85,B 0,C 180,E1 14132.296,E2 14132.296} C_VEL
LIN {X 0,Y 319.733,Z 958.75,A -85,B 0,C 180,E1 14128.561,E2 14128.561} C_VEL
LIN {X 0,Y 318.317,Z 962.79,A -85,B 0,C 180,E1 14126.915,E2 14126.915} C_VEL
LIN {X 0,Y 316.364,Z 965.918,A -85,B 0,C 180,E1 14125.679,E2 14125.679} C_VEL
LIN {X 0,Y 308.096,Z 973.672,A -85,B 0,C 180,E1 14122.376,E2 14122.376} C_VEL
LIN {X 0,Y 306.779,Z 975.735,A -85,B 0,C 180,E1 14121.219,E2 14121.219} C_VEL
LIN {X 0,Y 305.266,Z 981.733,A -85,B 0,C 180,E1 14117.126,E2 14117.126} C_VEL
LIN {X 0,Y 304.408,Z 986.561,A -85,B 0,C 180,E1 14112.8,E2 14112.8} C_VEL
LIN {X 0,Y 304.085,Z 989.391,A -85,B 0,C 180,E1 14108.993,E2 14108.993} C_VEL
LIN {X 0,Y 303.99,Z 991.096,A -85,B 0,C 180,E1 14105.205,E2 14105.205} C_VEL
LIN {X 0,Y 303.982,Z 991.53,A -85,B 0,C 180,E1 14101.038,E2 14101.038} C_VEL
LIN {X 0,Y 303.993,Z 990.807,A -85,B 0,C 180,E1 14097.575,E2 14097.575} C_VEL
LIN {X 0,Y 304.176,Z 988.765,A -85,B 0,C 180,E1 14093.484,E2 14093.484} C_VEL
LIN {X 0,Y 304.686,Z 985.258,A -85,B 0,C 180,E1 14089.471,E2 14089.471} C_VEL
LIN {X 0,Y 305.809,Z 980.174,A -85,B 0,C 180,E1 14085.195,E2 14085.195} C_VEL
LIN {X 0,Y 307.687,Z 973.478,A -85,B 0,C 180,E1 14081.028,E2 14081.028} C_VEL
LIN {X 0,Y 310.456,Z 965.499,A -85,B 0,C 180,E1 14076.986,E2 14076.986} C_VEL
LIN {X 0,Y 314.269,Z 955.563,A -85,B 0,C 180,E1 14072.96,E2 14072.96} C_VEL
LIN {X 0,Y 319.501,Z 943.092,A -85,B 0,C 180,E1 14068.8,E2 14068.8} C_VEL
LIN {X 0,Y 325.105,Z 930.331,A -85,B 0,C 180,E1 14065.277,E2 14065.277} C_VEL
LIN {X 0,Y 331.398,Z 915.867,A -85,B 0,C 180,E1 14061.971,E2 14061.971} C_VEL
LIN {X 0,Y 338.268,Z 900.045,A -85,B 0,C 180,E1 14058.93,E2 14058.93} C_VEL
LIN {X 0,Y 344.927,Z 883.969,A -85,B 0,C 180,E1 14056.355,E2 14056.355} C_VEL
LIN {X 0,Y 352.427,Z 864.841,A -85,B 0,C 180,E1 14053.788,E2 14053.788} C_VEL
LIN {X 0,Y 359.154,Z 846.359,A -85,B 0,C 180,E1 14051.726,E2 14051.726} C_VEL
LIN {X 0,Y 365.569,Z 826.819,A -85,B 0,C 180,E1 14049.923,E2 14049.923} C_VEL
LIN {X 0,Y 371.636,Z 806.344,A -85,B 0,C 180,E1 14048.354,E2 14048.354} C_VEL
LIN {X 0,Y 376.957,Z 785.213,A -85,B 0,C 180,E1 14047.051,E2 14047.051} C_VEL
LIN {X 0,Y 381.802,Z 762.511,A -85,B 0,C 180,E1 14045.933,E2 14045.933} C_VEL
LIN {X 0,Y 385.448,Z 740.812,A -85,B 0,C 180,E1 14045.114,E2 14045.114} C_VEL
LIN {X 0,Y 388.474,Z 716.359,A -85,B 0,C 180,E1 14044.445,E2 14044.445} C_VEL
LIN {X 0,Y 405.273,Z 505.838,A -85,B 0,C 180,E1 14040.107,E2 14040.107} C_VEL
LIN {X 0,Y 400.35,Z 497.23,A -85,B 0,C 180,E1 14037.782,E2 14037.782} C_VEL
LIN {X 0,Y 396.451,Z 490.47,A -85,B 0,C 180,E1 14035.516,E2 14035.516} C_VEL
LIN {X 0,Y 393.573,Z 485.81,A -85,B 0,C 180,E1 14033.393,E2 14033.393} C_VEL
LIN {X 0,Y 391.177,Z 481.578,A -85,B 0,C 180,E1 14030.882,E2 14030.882} C_VEL
LIN {X 0,Y 389.38,Z 478.948,A -85,B 0,C 180,E1 14026.487,E2 14026.487} C_VEL
LIN {X 0,Y 389.651,Z 479.813,A -85,B 0,C 180,E1 14024.217,E2 14024.217} C_VEL
LIN {X 0,Y 391.441,Z 481.989,A -85,B 0,C 180,E1 14021.226,E2 14021.226} C_VEL
LIN {X 0,Y 393.795,Z 486.109,A -85,B 0,C 180,E1 14018.867,E2 14018.867} C_VEL
LIN {X 0,Y 397.116,Z 491.852,A -85,B 0,C 180,E1 14016.481,E2 14016.481} C_VEL
LIN {X 0,Y 401.383,Z 500.223,A -85,B 0,C 180,E1 14014.066,E2 14014.066} C_VEL
LIN {X 0,Y 405.195,Z 508.331,A -85,B 0,C 180,E1 14012.241,E2 14012.241} C_VEL
LIN {X 0,Y 390.136,Z 698.968,A -85,B 0,C 180,E1 14008.319,E2 14008.319} C_VEL
LIN {X 0,Y 387.033,Z 736.287,A -85,B 0,C 180,E1 14007.514,E2 14007.514} C_VEL
LIN {X 0,Y 383.795,Z 758.936,A -85,B 0,C 180,E1 14006.87,E2 14006.87} C_VEL
LIN {X 0,Y 379.394,Z 782.33,A -85,B 0,C 180,E1 14005.984,E2 14005.984} C_VEL
LIN {X 0,Y 374.791,Z 802.536,A -85,B 0,C 180,E1 14004.99,E2 14004.99} C_VEL
LIN {X 0,Y 368.887,Z 824.723,A -85,B 0,C 180,E1 14003.616,E2 14003.616} C_VEL
LIN {X 0,Y 363.245,Z 843.578,A -85,B 0,C 180,E1 14002.189,E2 14002.189} C_VEL
LIN {X 0,Y 356.281,Z 864.497,A -85,B 0,C 180,E1 14000.264,E2 14000.264} C_VEL
LIN {X 0,Y 349.648,Z 883.012,A -85,B 0,C 180,E1 13998.22,E2 13998.22} C_VEL
LIN {X 0,Y 342.324,Z 901.945,A -85,B 0,C 180,E1 13995.697,E2 13995.697} C_VEL
LIN {X 0,Y 335.47,Z 919.191,A -85,B 0,C 180,E1 13992.963,E2 13992.963} C_VEL
LIN {X 0,Y 328.857,Z 935.224,A -85,B 0,C 180,E1 13989.911,E2 13989.911} C_VEL
LIN {X 0,Y 322.399,Z 950.994,A -85,B 0,C 180,E1 13986.329,E2 13986.329} C_VEL
LIN {X 0,Y 317.266,Z 963.938,A -85,B 0,C 180,E1 13982.829,E2 13982.829} C_VEL
LIN {X 0,Y 312.708,Z 976.075,A -85,B 0,C 180,E1 13978.874,E2 13978.874} C_VEL
LIN {X 0,Y 309.264,Z 986.42,A -85,B 0,C 180,E1 13974.858,E2 13974.858} C_VEL
LIN {X 0,Y 306.759,Z 995.058,A -85,B 0,C 180,E1 13970.701,E2 13970.701} C_VEL
LIN {X 0,Y 305.14,Z 1002.328,A -85,B 0,C 180,E1 13966.373,E2 13966.373} C_VEL
LIN {X 0,Y 304.355,Z 1007.261,A -85,B 0,C 180,E1 13962.528,E2 13962.528} C_VEL
LIN {X 0,Y 304.035,Z 1011.12,A -85,B 0,C 180,E1 13958.516,E2 13958.516} C_VEL
LIN {X 0,Y 303.955,Z 1013.39,A -85,B 0,C 180,E1 13954.534,E2 13954.534} C_VEL
LIN {X 0,Y 303.963,Z 1014.275,A -85,B 0,C 180,E1 13951.137,E2 13951.137} C_VEL
LIN {X 0,Y 303.954,Z 1014.11,A -85,B 0,C 180,E1 13947.366,E2 13947.366} C_VEL
LIN {X 0,Y 303.973,Z 1012.418,A -85,B 0,C 180,E1 13943.391,E2 13943.391} C_VEL
LIN {X 0,Y 304.091,Z 1009.892,A -85,B 0,C 180,E1 13939.97,E2 13939.97} C_VEL
LIN {X 0,Y 304.639,Z 1005.4,A -85,B 0,C 180,E1 13935.756,E2 13935.756} C_VEL
LIN {X 0,Y 305.673,Z 999.78,A -85,B 0,C 180,E1 13931.903,E2 13931.903} C_VEL
LIN {X 0,Y 307.521,Z 992.461,A -85,B 0,C 180,E1 13927.849,E2 13927.849} C_VEL
LIN {X 0,Y 310.288,Z 983.279,A -85,B 0,C 180,E1 13923.81,E2 13923.81} C_VEL
LIN {X 0,Y 314.105,Z 972.372,A -85,B 0,C 180,E1 13919.813,E2 13919.813} C_VEL
LIN {X 0,Y 318.51,Z 960.636,A -85,B 0,C 180,E1 13916.254,E2 13916.254} C_VEL
LIN {X 0,Y 324.169,Z 946.249,A -85,B 0,C 180,E1 13912.591,E2 13912.591} C_VEL
LIN {X 0,Y 329.915,Z 931.905,A -85,B 0,C 180,E1 13909.524,E2 13909.524} C_VEL
LIN {X 0,Y 336.445,Z 915.257,A -85,B 0,C 180,E1 13906.539,E2 13906.539} C_VEL
LIN {X 0,Y 343.147,Z 897.817,A -85,B 0,C 180,E1 13903.905,E2 13903.905} C_VEL
LIN {X 0,Y 349.691,Z 879.533,A -85,B 0,C 180,E1 13901.619,E2 13901.619} C_VEL
LIN {X 0,Y 356.186,Z 860.255,A -85,B 0,C 180,E1 13899.584,E2 13899.584} C_VEL
LIN {X 0,Y 362.002,Z 841.128,A -85,B 0,C 180,E1 13897.917,E2 13897.917} C_VEL
LIN {X 0,Y 367.899,Z 819.525,A -85,B 0,C 180,E1 13896.361,E2 13896.361} C_VEL
LIN {X 0,Y 372.587,Z 799.735,A -85,B 0,C 180,E1 13895.212,E2 13895.212} C_VEL
LIN {X 0,Y 377.381,Z 775.629,A -85,B 0,C 180,E1 13894.104,E2 13894.104} C_VEL
LIN {X 0,Y 380.947,Z 753.349,A -85,B 0,C 180,E1 13893.339,E2 13893.339} C_VEL
LIN {X 0,Y 383.51,Z 729.705,A -85,B 0,C 180,E1 13892.744,E2 13892.744} C_VEL
LIN {X 0,Y 397.013,Z 523.038,A -85,B 0,C 180,E1 13888.603,E2 13888.603} C_VEL
LIN {X 0,Y 398.05,Z 506.652,A -85,B 0,C 180,E1 13888.261,E2 13888.261} C_VEL
LIN {X 0,Y 389.357,Z 492.524,A -85,B 0,C 180,E1 13885.516,E2 13885.516} C_VEL
LIN {X 0,Y 381.9,Z 481.048,A -85,B 0,C 180,E1 13882.919,E2 13882.919} C_VEL
LIN {X 0,Y 374.824,Z 471.006,A -85,B 0,C 180,E1 13880.208,E2 13880.208} C_VEL
LIN {X 0,Y 371.163,Z 466.269,A -85,B 0,C 180,E1 13878.697,E2 13878.697} C_VEL
LIN {X 0,Y 368,Z 462.195,A -85,B 0,C 180,E1 13877.308,E2 13877.308} C_VEL
LIN {X 0,Y 363.886,Z 457.011,A -85,B 0,C 180,E1 13875.376,E2 13875.376} C_VEL
LIN {X 0,Y 359.622,Z 451.708,A -85,B 0,C 180,E1 13873.178,E2 13873.178} C_VEL
LIN {X 0,Y 356.017,Z 447.417,A -85,B 0,C 180,E1 13871.132,E2 13871.132} C_VEL
LIN {X 0,Y 355.064,Z 446.076,A -85,B 0,C 180,E1 13870.546,E2 13870.546} C_VEL
LIN {X 0,Y 351.482,Z 442.319,A -85,B 0,C 180,E1 13868.259,E2 13868.259} C_VEL
LIN {X 0,Y 350.08,Z 440.094,A -85,B 0,C 180,E1 13867.219,E2 13867.219} C_VEL
LIN {X 0,Y 346.659,Z 436.976,A -85,B 0,C 180,E1 13864.632,E2 13864.632} C_VEL
LIN {X 0,Y 344.917,Z 433.892,A -85,B 0,C 180,E1 13862.99,E2 13862.99} C_VEL
LIN {X 0,Y 341.279,Z 431.102,A -85,B 0,C 180,E1 13859.328,E2 13859.328} C_VEL
LIN {X 0,Y 339.327,Z 427.473,A -85,B 0,C 180,E1 13856.452,E2 13856.452} C_VEL
LIN {X 0,Y 335.987,Z 425.386,A -85,B 0,C 180,E1 13849.02,E2 13849.02} C_VEL
LIN {X 0,Y 335.71,Z 425.112,A -85,B 0,C 180,E1 13844.096,E2 13844.096} C_VEL
LIN {X 0,Y 337.387,Z 426.49,A -85,B 0,C 180,E1 13838.042,E2 13838.042} C_VEL
LIN {X 0,Y 339.595,Z 427.767,A -85,B 0,C 180,E1 13834.353,E2 13834.353} C_VEL
LIN {X 0,Y 341.779,Z 431.616,A -85,B 0,C 180,E1 13831.329,E2 13831.329} C_VEL
LIN {X 0,Y 345.132,Z 434.148,A -85,B 0,C 180,E1 13828.071,E2 13828.071} C_VEL
LIN {X 0,Y 347.57,Z 438.029,A -85,B 0,C 180,E1 13825.877,E2 13825.877} C_VEL
LIN {X 0,Y 350.53,Z 440.666,A -85,B 0,C 180,E1 13823.709,E2 13823.709} C_VEL
LIN {X 0,Y 353.417,Z 444.655,A -85,B 0,C 180,E1 13821.714,E2 13821.714} C_VEL
LIN {X 0,Y 355.694,Z 446.867,A -85,B 0,C 180,E1 13820.349,E2 13820.349} C_VEL
LIN {X 0,Y 359.249,Z 451.342,A -85,B 0,C 180,E1 13818.303,E2 13818.303} C_VEL
LIN {X 0,Y 360.829,Z 453.143,A -85,B 0,C 180,E1 13817.474,E2 13817.474} C_VEL
LIN {X 0,Y 365.64,Z 459.167,A -85,B 0,C 180,E1 13815.083,E2 13815.083} C_VEL
LIN {X 0,Y 370.215,Z 464.999,A -85,B 0,C 180,E1 13813.015,E2 13813.015} C_VEL
LIN {X 0,Y 374.833,Z 470.992,A -85,B 0,C 180,E1 13811.099,E2 13811.099} C_VEL
LIN {X 0,Y 381.171,Z 479.224,A -85,B 0,C 180,E1 13808.704,E2 13808.704} C_VEL
LIN {X 0,Y 391.054,Z 493.081,A -85,B 0,C 180,E1 13805.349,E2 13805.349} C_VEL
LIN {X 0,Y 397.785,Z 503.349,A -85,B 0,C 180,E1 13803.272,E2 13803.272} C_VEL
LIN {X 0,Y 384.116,Z 711.172,A -85,B 0,C 180,E1 13799.116,E2 13799.116} C_VEL
LIN {X 0,Y 381.706,Z 734.593,A -85,B 0,C 180,E1 13798.52,E2 13798.52} C_VEL
LIN {X 0,Y 378.393,Z 756.475,A -85,B 0,C 180,E1 13797.74,E2 13797.74} C_VEL
LIN {X 0,Y 374.333,Z 778.201,A -85,B 0,C 180,E1 13796.742,E2 13796.742} C_VEL
LIN {X 0,Y 369.666,Z 798.635,A -85,B 0,C 180,E1 13795.551,E2 13795.551} C_VEL
LIN {X 0,Y 364.157,Z 819.639,A -85,B 0,C 180,E1 13794.056,E2 13794.056} C_VEL
LIN {X 0,Y 358.599,Z 838.167,A -85,B 0,C 180,E1 13792.451,E2 13792.451} C_VEL
LIN {X 0,Y 351.972,Z 858.213,A -85,B 0,C 180,E1 13790.372,E2 13790.372} C_VEL
LIN {X 0,Y 345.678,Z 875.69,A -85,B 0,C 180,E1 13788.197,E2 13788.197} C_VEL
LIN {X 0,Y 338.894,Z 893.373,A -85,B 0,C 180,E1 13785.568,E2 13785.568} C_VEL
LIN {X 0,Y 332.709,Z 908.817,A -85,B 0,C 180,E1 13782.843,E2 13782.843} C_VEL
LIN {X 0,Y 326.492,Z 923.754,A -85,B 0,C 180,E1 13779.691,E2 13779.691} C_VEL
LIN {X 0,Y 320.858,Z 937.486,A -85,B 0,C 180,E1 13776.256,E2 13776.256} C_VEL
LIN {X 0,Y 316.072,Z 949.183,A -85,B 0,C 180,E1 13772.714,E2 13772.714} C_VEL
LIN {X 0,Y 311.842,Z 960.242,A -85,B 0,C 180,E1 13768.708,E2 13768.708} C_VEL
LIN {X 0,Y 308.902,Z 968.664,A -85,B 0,C 180,E1 13764.981,E2 13764.981} C_VEL
LIN {X 0,Y 306.779,Z 975.735,A -85,B 0,C 180,E1 13761.219,E2 13761.219} C_VEL
LIN {X 0,Y 305.196,Z 977.991,A -85,B 0,C 180,E1 13759.859,E2 13759.859} C_VEL
LIN {X 0,Y 299.493,Z 982.228,A -85,B 0,C 180,E1 13757.207,E2 13757.207} C_VEL
LIN {X 0,Y 297.012,Z 984.41,A -85,B 0,C 180,E1 13755.496,E2 13755.496} C_VEL
LIN {X 0,Y 296.764,Z 984.957,A -85,B 0,C 180,E1 13754.971,E2 13754.971} C_VEL
LIN {X 0,Y 296.218,Z 988.451,A -85,B 0,C 180,E1 13751.087,E2 13751.087} C_VEL
LIN {X 0,Y 296.007,Z 990.816,A -85,B 0,C 180,E1 13746.926,E2 13746.926} C_VEL
LIN {X 0,Y 295.968,Z 991.752,A -85,B 0,C 180,E1 13743.295,E2 13743.295} C_VEL
LIN {X 0,Y 295.978,Z 991.686,A -85,B 0,C 180,E1 13739.549,E2 13739.549} C_VEL
LIN {X 0,Y 296.066,Z 990.293,A -85,B 0,C 180,E1 13735.428,E2 13735.428} C_VEL
LIN {X 0,Y 296.369,Z 987.818,A -85,B 0,C 180,E1 13731.623,E2 13731.623} C_VEL
LIN {X 0,Y 297.148,Z 983.863,A -85,B 0,C 180,E1 13727.436,E2 13727.436} C_VEL
LIN {X 0,Y 298.689,Z 978.053,A -85,B 0,C 180,E1 13723.071,E2 13723.071} C_VEL
LIN {X 0,Y 301.244,Z 970.477,A -85,B 0,C 180,E1 13718.609,E2 13718.609} C_VEL
LIN {X 0,Y 304.639,Z 961.749,A -85,B 0,C 180,E1 13714.525,E2 13714.525} C_VEL
LIN {X 0,Y 309.432,Z 950.583,A -85,B 0,C 180,E1 13710.271,E2 13710.271} C_VEL
LIN {X 0,Y 314.983,Z 938.493,A -85,B 0,C 180,E1 13706.463,E2 13706.463} C_VEL
LIN {X 0,Y 321.138,Z 925.049,A -85,B 0,C 180,E1 13702.992,E2 13702.992} C_VEL
LIN {X 0,Y 328.174,Z 909.833,A -85,B 0,C 180,E1 13699.696,E2 13699.696} C_VEL
LIN {X 0,Y 335.065,Z 894.369,A -85,B 0,C 180,E1 13696.906,E2 13696.906} C_VEL
LIN {X 0,Y 342.76,Z 876.276,A -85,B 0,C 180,E1 13694.185,E2 13694.185} C_VEL
LIN {X 0,Y 350.192,Z 857.732,A -85,B 0,C 180,E1 13691.864,E2 13691.864} C_VEL
LIN {X 0,Y 356.998,Z 838.85,A -85,B 0,C 180,E1 13689.919,E2 13689.919} C_VEL
LIN {X 0,Y 363.667,Z 818.651,A -85,B 0,C 180,E1 13688.182,E2 13688.182} C_VEL
LIN {X 0,Y 369.328,Z 798.886,A -85,B 0,C 180,E1 13686.798,E2 13686.798} C_VEL
LIN {X 0,Y 374.726,Z 777.241,A -85,B 0,C 180,E1 13685.561,E2 13685.561} C_VEL
LIN {X 0,Y 378.894,Z 756.834,A -85,B 0,C 180,E1 13684.641,E2 13684.641} C_VEL
LIN {X 0,Y 382.642,Z 733.775,A -85,B 0,C 180,E1 13683.845,E2 13683.845} C_VEL
LIN {X 0,Y 385.158,Z 711.61,A -85,B 0,C 180,E1 13683.287,E2 13683.287} C_VEL
LIN {X 0,Y 401.872,Z 510.785,A -85,B 0,C 180,E1 13679.145,E2 13679.145} C_VEL
LIN {X 0,Y 397.468,Z 502.794,A -85,B 0,C 180,E1 13676.868,E2 13676.868} C_VEL
LIN {X 0,Y 394.278,Z 497.226,A -85,B 0,C 180,E1 13674.836,E2 13674.836} C_VEL
LIN {X 0,Y 392.207,Z 493.572,A -85,B 0,C 180,E1 13673.193,E2 13673.193} C_VEL
LIN {X 0,Y 389.935,Z 489.414,A -85,B 0,C 180,E1 13670.704,E2 13670.704} C_VEL
LIN {X 0,Y 388.291,Z 486.87,A -85,B 0,C 180,E1 13666.449,E2 13666.449} C_VEL
LIN {X 0,Y 388.575,Z 487.795,A -85,B 0,C 180,E1 13664.172,E2 13664.172} C_VEL
LIN {X 0,Y 390.186,Z 489.879,A -85,B 0,C 180,E1 13661.396,E2 13661.396} C_VEL
LIN {X 0,Y 392.896,Z 494.825,A -85,B 0,C 180,E1 13658.66,E2 13658.66} C_VEL
LIN {X 0,Y 395.651,Z 499.761,A -85,B 0,C 180,E1 13656.664,E2 13656.664} C_VEL
LIN {X 0,Y 399.847,Z 508.542,A -85,B 0,C 180,E1 13654.209,E2 13654.209} C_VEL
LIN {X 0,Y 401.804,Z 513.104,A -85,B 0,C 180,E1 13653.203,E2 13653.203} C_VEL
LIN {X 0,Y 385.981,Z 704.664,A -85,B 0,C 180,E1 13649.252,E2 13649.252} C_VEL
LIN {X 0,Y 382.968,Z 737.575,A -85,B 0,C 180,E1 13648.525,E2 13648.525} C_VEL
LIN {X 0,Y 379.538,Z 760.458,A -85,B 0,C 180,E1 13647.868,E2 13647.868} C_VEL
LIN {X 0,Y 375.006,Z 783.242,A -85,B 0,C 180,E1 13646.991,E2 13646.991} C_VEL
LIN {X 0,Y 369.959,Z 804.437,A -85,B 0,C 180,E1 13645.935,E2 13645.935} C_VEL
LIN {X 0,Y 364.167,Z 825.123,A -85,B 0,C 180,E1 13644.636,E2 13644.636} C_VEL
LIN {X 0,Y 357.771,Z 845.609,A -85,B 0,C 180,E1 13643.066,E2 13643.066} C_VEL
LIN {X 0,Y 350.846,Z 865.334,A -85,B 0,C 180,E1 13641.214,E2 13641.214} C_VEL
LIN {X 0,Y 343.851,Z 884.01,A -85,B 0,C 180,E1 13639.121,E2 13639.121} C_VEL
LIN {X 0,Y 336.426,Z 902.273,A -85,B 0,C 180,E1 13636.645,E2 13636.645} C_VEL
LIN {X 0,Y 328.942,Z 920.097,A -85,B 0,C 180,E1 13633.755,E2 13633.755} C_VEL
LIN {X 0,Y 322.419,Z 935.19,A -85,B 0,C 180,E1 13630.829,E2 13630.829} C_VEL
LIN {X 0,Y 315.675,Z 950.757,A -85,B 0,C 180,E1 13627.232,E2 13627.232} C_VEL
LIN {X 0,Y 310.253,Z 963.673,A -85,B 0,C 180,E1 13623.668,E2 13623.668} C_VEL
LIN {X 0,Y 305.603,Z 975.263,A -85,B 0,C 180,E1 13619.827,E2 13619.827} C_VEL
LIN {X 0,Y 301.847,Z 985.703,A -85,B 0,C 180,E1 13615.713,E2 13615.713} C_VEL
LIN {X 0,Y 299.171,Z 994.18,A -85,B 0,C 180,E1 13611.575,E2 13611.575} C_VEL
LIN {X 0,Y 297.379,Z 1001.489,A -85,B 0,C 180,E1 13607.216,E2 13607.216} C_VEL
LIN {X 0,Y 296.435,Z 1006.743,A -85,B 0,C 180,E1 13603.066,E2 13603.066} C_VEL
LIN {X 0,Y 296.047,Z 1010.655,A -85,B 0,C 180,E1 13598.943,E2 13598.943} C_VEL
LIN {X 0,Y 295.958,Z 1013.017,A -85,B 0,C 180,E1 13594.851,E2 13594.851} C_VEL
LIN {X 0,Y 295.973,Z 1013.951,A -85,B 0,C 180,E1 13591.361,E2 13591.361} C_VEL
LIN {X 0,Y 295.968,Z 1013.855,A -85,B 0,C 180,E1 13587.683,E2 13587.683} C_VEL
LIN {X 0,Y 295.977,Z 1012.346,A -85,B 0,C 180,E1 13583.606,E2 13583.606} C_VEL
LIN {X 0,Y 296.085,Z 1009.908,A -85,B 0,C 180,E1 13580.089,E2 13580.089} C_VEL
LIN {X 0,Y 296.565,Z 1006.01,A -85,B 0,C 180,E1 13576.157,E2 13576.157} C_VEL
LIN {X 0,Y 297.694,Z 1000.059,A -85,B 0,C 180,E1 13571.806,E2 13571.806} C_VEL
LIN {X 0,Y 299.491,Z 993.209,A -85,B 0,C 180,E1 13567.844,E2 13567.844} C_VEL
LIN {X 0,Y 302.476,Z 983.844,A -85,B 0,C 180,E1 13563.504,E2 13563.504} C_VEL
LIN {X 0,Y 306.338,Z 973.388,A -85,B 0,C 180,E1 13559.503,E2 13559.503} C_VEL
LIN {X 0,Y 311.274,Z 960.841,A -85,B 0,C 180,E1 13555.583,E2 13555.583} C_VEL
LIN {X 0,Y 317.203,Z 946.555,A -85,B 0,C 180,E1 13551.852,E2 13551.852} C_VEL
LIN {X 0,Y 323.151,Z 932.323,A -85,B 0,C 180,E1 13548.751,E2 13548.751} C_VEL
LIN {X 0,Y 330.231,Z 915.068,A -85,B 0,C 180,E1 13545.605,E2 13545.605} C_VEL
LIN {X 0,Y 337.256,Z 897.533,A -85,B 0,C 180,E1 13542.932,E2 13542.932} C_VEL
LIN {X 0,Y 343.953,Z 879.495,A -85,B 0,C 180,E1 13540.659,E2 13540.659} C_VEL
LIN {X 0,Y 350.819,Z 859.756,A -85,B 0,C 180,E1 13538.569,E2 13538.569} C_VEL
LIN {X 0,Y 356.866,Z 840.487,A -85,B 0,C 180,E1 13536.89,E2 13536.89} C_VEL
LIN {X 0,Y 363.112,Z 818.188,A -85,B 0,C 180,E1 13535.296,E2 13535.296} C_VEL
LIN {X 0,Y 368.202,Z 797.217,A -85,B 0,C 180,E1 13534.094,E2 13534.094} C_VEL
LIN {X 0,Y 372.879,Z 773.9,A -85,B 0,C 180,E1 13533.052,E2 13533.052} C_VEL
LIN {X 0,Y 376.622,Z 750.81,A -85,B 0,C 180,E1 13532.281,E2 13532.281} C_VEL
LIN {X 0,Y 379.086,Z 727.382,A -85,B 0,C 180,E1 13531.707,E2 13531.707} C_VEL
LIN {X 0,Y 393.216,Z 518.434,A -85,B 0,C 180,E1 13527.511,E2 13527.511} C_VEL
LIN {X 0,Y 393.643,Z 510.752,A -85,B 0,C 180,E1 13527.329,E2 13527.329} C_VEL
LIN {X 0,Y 383.788,Z 494.782,A -85,B 0,C 180,E1 13524.061,E2 13524.061} C_VEL
LIN {X 0,Y 375.884,Z 482.827,A -85,B 0,C 180,E1 13521.126,E2 13521.126} C_VEL
LIN {X 0,Y 369.91,Z 474.64,A -85,B 0,C 180,E1 13518.681,E2 13518.681} C_VEL
LIN {X 0,Y 365.623,Z 469.143,A -85,B 0,C 180,E1 13516.768,E2 13516.768} C_VEL
LIN {X 0,Y 362.041,Z 464.512,A -85,B 0,C 180,E1 13515.046,E2 13515.046} C_VEL
LIN {X 0,Y 357.839,Z 459.242,A -85,B 0,C 180,E1 13512.842,E2 13512.842} C_VEL
LIN {X 0,Y 354.143,Z 454.714,A -85,B 0,C 180,E1 13510.697,E2 13510.697} C_VEL
LIN {X 0,Y 352.807,Z 453.211,A -85,B 0,C 180,E1 13509.872,E2 13509.872} C_VEL
LIN {X 0,Y 349.379,Z 449.109,A -85,B 0,C 180,E1 13507.564,E2 13507.564} C_VEL
LIN {X 0,Y 348.342,Z 447.669,A -85,B 0,C 180,E1 13506.779,E2 13506.779} C_VEL
LIN {X 0,Y 345.007,Z 444.339,A -85,B 0,C 180,E1 13504.154,E2 13504.154} C_VEL
LIN {X 0,Y 343.452,Z 441.651,A -85,B 0,C 180,E1 13502.669,E2 13502.669} C_VEL
LIN {X 0,Y 339.911,Z 438.759,A -85,B 0,C 180,E1 13498.988,E2 13498.988} C_VEL
LIN {X 0,Y 338.116,Z 435.325,A -85,B 0,C 180,E1 13496.269,E2 13496.269} C_VEL
LIN {X 0,Y 334.869,Z 433.262,A -85,B 0,C 180,E1 13488.808,E2 13488.808} C_VEL
LIN {X 0,Y 334.654,Z 433.083,A -85,B 0,C 180,E1 13483.867,E2 13483.867} C_VEL
LIN {X 0,Y 336.416,Z 434.494,A -85,B 0,C 180,E1 13477.823,E2 13477.823} C_VEL
LIN {X 0,Y 338.436,Z 435.718,A -85,B 0,C 180,E1 13474.447,E2 13474.447} C_VEL
LIN {X 0,Y 340.453,Z 439.365,A -85,B 0,C 180,E1 13471.59,E2 13471.59} C_VEL
LIN {X 0,Y 343.828,Z 442.131,A -85,B 0,C 180,E1 13468.24,E2 13468.24} C_VEL
LIN {X 0,Y 346.391,Z 446.02,A -85,B 0,C 180,E1 13465.925,E2 13465.925} C_VEL
LIN {X 0,Y 349.009,Z 448.405,A -85,B 0,C 180,E1 13463.983,E2 13463.983} C_VEL
LIN {X 0,Y 352.044,Z 452.504,A -85,B 0,C 180,E1 13461.869,E2 13461.869} C_VEL
LIN {X 0,Y 354.017,Z 454.495,A -85,B 0,C 180,E1 13460.659,E2 13460.659} C_VEL
LIN {X 0,Y 357.73,Z 459.11,A -85,B 0,C 180,E1 13458.499,E2 13458.499} C_VEL
LIN {X 0,Y 360.237,Z 462.403,A -85,B 0,C 180,E1 13457.155,E2 13457.155} C_VEL
LIN {X 0,Y 363.612,Z 466.497,A -85,B 0,C 180,E1 13455.476,E2 13455.476} C_VEL
LIN {X 0,Y 368.303,Z 472.579,A -85,B 0,C 180,E1 13453.317,E2 13453.317} C_VEL
LIN {X 0,Y 375.227,Z 481.505,A -85,B 0,C 180,E1 13450.467,E2 13450.467} C_VEL
LIN {X 0,Y 383.454,Z 493.008,A -85,B 0,C 180,E1 13447.439,E2 13447.439} C_VEL
LIN {X 0,Y 391.217,Z 504.289,A -85,B 0,C 180,E1 13444.874,E2 13444.874} C_VEL
LIN {X 0,Y 393.386,Z 507.873,A -85,B 0,C 180,E1 13444.184,E2 13444.184} C_VEL
LIN {X 0,Y 379.331,Z 713.863,A -85,B 0,C 180,E1 13440.047,E2 13440.047} C_VEL
LIN {X 0,Y 376.444,Z 738.904,A -85,B 0,C 180,E1 13439.375,E2 13439.375} C_VEL
LIN {X 0,Y 373.071,Z 760.075,A -85,B 0,C 180,E1 13438.59,E2 13438.59} C_VEL
LIN {X 0,Y 368.655,Z 781.965,A -85,B 0,C 180,E1 13437.537,E2 13437.537} C_VEL
LIN {X 0,Y 363.628,Z 803.025,A -85,B 0,C 180,E1 13436.27,E2 13436.27} C_VEL
LIN {X 0,Y 357.946,Z 823.241,A -85,B 0,C 180,E1 13434.765,E2 13434.765} C_VEL
LIN {X 0,Y 351.777,Z 842.997,A -85,B 0,C 180,E1 13432.999,E2 13432.999} C_VEL
LIN {X 0,Y 344.949,Z 862.408,A -85,B 0,C 180,E1 13430.881,E2 13430.881} C_VEL
LIN {X 0,Y 337.756,Z 881.394,A -85,B 0,C 180,E1 13428.389,E2 13428.389} C_VEL
LIN {X 0,Y 331.404,Z 897.063,A -85,B 0,C 180,E1 13425.929,E2 13425.929} C_VEL
LIN {X 0,Y 324.353,Z 913.706,A -85,B 0,C 180,E1 13422.818,E2 13422.818} C_VEL
LIN {X 0,Y 318.425,Z 927.432,A -85,B 0,C 180,E1 13419.756,E2 13419.756} C_VEL
LIN {X 0,Y 312.677,Z 940.594,A -85,B 0,C 180,E1 13416.236,E2 13416.236} C_VEL
LIN {X 0,Y 307.672,Z 952.576,A -85,B 0,C 180,E1 13412.416,E2 13412.416} C_VEL
LIN {X 0,Y 303.618,Z 962.614,A -85,B 0,C 180,E1 13408.485,E2 13408.485} C_VEL
LIN {X 0,Y 300.44,Z 971.519,A -85,B 0,C 180,E1 13404.264,E2 13404.264} C_VEL
LIN {X 0,Y 298.308,Z 978.389,A -85,B 0,C 180,E1 13400.152,E2 13400.152} C_VEL
LIN {X 0,Y 296.925,Z 984.137,A -85,B 0,C 180,E1 13395.764,E2 13395.764} C_VEL
LIN {X 0,Y 296.764,Z 984.957,A -85,B 0,C 180,E1 13394.971,E2 13394.971} C_VEL
LIN {X 0,Y 295.528,Z 986.539,A -85,B 0,C 180,E1 13393.518,E2 13393.518} C_VEL
LIN {X 0,Y 288.766,Z 989.88,A -85,B 0,C 180,E1 13389.492,E2 13389.492} C_VEL
LIN {X 0,Y 288.06,Z 990.576,A -85,B 0,C 180,E1 13388.287,E2 13388.287} C_VEL
LIN {X 0,Y 287.97,Z 991.961,A -85,B 0,C 180,E1 13384.051,E2 13384.051} C_VEL
LIN {X 0,Y 287.977,Z 992.085,A -85,B 0,C 180,E1 13380.455,E2 13380.455} C_VEL
LIN {X 0,Y 288.03,Z 991.257,A -85,B 0,C 180,E1 13376.784,E2 13376.784} C_VEL
LIN {X 0,Y 288.296,Z 988.935,A -85,B 0,C 180,E1 13372.376,E2 13372.376} C_VEL
LIN {X 0,Y 288.937,Z 985.52,A -85,B 0,C 180,E1 13368.357,E2 13368.357} C_VEL
LIN {X 0,Y 290.384,Z 980.215,A -85,B 0,C 180,E1 13363.797,E2 13363.797} C_VEL
LIN {X 0,Y 292.683,Z 973.49,A -85,B 0,C 180,E1 13359.454,E2 13359.454} C_VEL
LIN {X 0,Y 296.389,Z 964.315,A -85,B 0,C 180,E1 13354.759,E2 13354.759} C_VEL
LIN {X 0,Y 300.942,Z 954.298,A -85,B 0,C 180,E1 13350.619,E2 13350.619} C_VEL
LIN {X 0,Y 306.34,Z 942.876,A -85,B 0,C 180,E1 13346.771,E2 13346.771} C_VEL
LIN {X 0,Y 312.886,Z 929.525,A -85,B 0,C 180,E1 13343.016,E2 13343.016} C_VEL
LIN {X 0,Y 319.534,Z 915.796,A -85,B 0,C 180,E1 13339.838,E2 13339.838} C_VEL
LIN {X 0,Y 327.574,Z 898.872,A -85,B 0,C 180,E1 13336.568,E2 13336.568} C_VEL
LIN {X 0,Y 335.142,Z 882.194,A -85,B 0,C 180,E1 13333.897,E2 13333.897} C_VEL
LIN {X 0,Y 342.831,Z 863.947,A -85,B 0,C 180,E1 13331.482,E2 13331.482} C_VEL
LIN {X 0,Y 350.395,Z 844.703,A -85,B 0,C 180,E1 13329.361,E2 13329.361} C_VEL
LIN {X 0,Y 357.12,Z 825.441,A -85,B 0,C 180,E1 13327.62,E2 13327.62} C_VEL
LIN {X 0,Y 363.965,Z 803.494,A -85,B 0,C 180,E1 13325.993,E2 13325.993} C_VEL
LIN {X 0,Y 369.005,Z 784.664,A -85,B 0,C 180,E1 13324.858,E2 13324.858} C_VEL
LIN {X 0,Y 374.246,Z 761.392,A -85,B 0,C 180,E1 13323.739,E2 13323.739} C_VEL
LIN {X 0,Y 377.936,Z 740.822,A -85,B 0,C 180,E1 13322.977,E2 13322.977} C_VEL
LIN {X 0,Y 381.078,Z 716.828,A -85,B 0,C 180,E1 13322.329,E2 13322.329} C_VEL
LIN {X 0,Y 398.638,Z 515.791,A -85,B 0,C 180,E1 13318.168,E2 13318.168} C_VEL
LIN {X 0,Y 394.615,Z 508.286,A -85,B 0,C 180,E1 13315.86,E2 13315.86} C_VEL
LIN {X 0,Y 392.378,Z 504.273,A -85,B 0,C 180,E1 13314.297,E2 13314.297} C_VEL
LIN {X 0,Y 390.62,Z 501.043,A -85,B 0,C 180,E1 13312.795,E2 13312.795} C_VEL
LIN {X 0,Y 388.696,Z 497.249,A -85,B 0,C 180,E1 13310.525,E2 13310.525} C_VEL
LIN {X 0,Y 387.202,Z 494.792,A -85,B 0,C 180,E1 13306.41,E2 13306.41} C_VEL
LIN {X 0,Y 387.552,Z 495.867,A -85,B 0,C 180,E1 13303.976,E2 13303.976} C_VEL
LIN {X 0,Y 388.883,Z 497.607,A -85,B 0,C 180,E1 13301.642,E2 13301.642} C_VEL
LIN {X 0,Y 391.461,Z 502.586,A -85,B 0,C 180,E1 13298.892,E2 13298.892} C_VEL
LIN {X 0,Y 393.926,Z 507.167,A -85,B 0,C 180,E1 13297.031,E2 13297.031} C_VEL
LIN {X 0,Y 397.938,Z 516.009,A -85,B 0,C 180,E1 13294.555,E2 13294.555} C_VEL
LIN {X 0,Y 398.576,Z 517.912,A -85,B 0,C 180,E1 13294.183,E2 13294.183} C_VEL
LIN {X 0,Y 381.949,Z 710.548,A -85,B 0,C 180,E1 13290.203,E2 13290.203} C_VEL
LIN {X 0,Y 378.963,Z 739.776,A -85,B 0,C 180,E1 13289.54,E2 13289.54} C_VEL
LIN {X 0,Y 375.213,Z 763.325,A -85,B 0,C 180,E1 13288.847,E2 13288.847} C_VEL
LIN {X 0,Y 370.745,Z 784.292,A -85,B 0,C 180,E1 13288.019,E2 13288.019} C_VEL
LIN {X 0,Y 365.235,Z 806.396,A -85,B 0,C 180,E1 13286.903,E2 13286.903} C_VEL
LIN {X 0,Y 359.191,Z 826.857,A -85,B 0,C 180,E1 13285.593,E2 13285.593} C_VEL
LIN {X 0,Y 352.378,Z 847.575,A -85,B 0,C 180,E1 13283.972,E2 13283.972} C_VEL
LIN {X 0,Y 345.518,Z 866.226,A -85,B 0,C 180,E1 13282.191,E2 13282.191} C_VEL
LIN {X 0,Y 337.743,Z 885.891,A -85,B 0,C 180,E1 13279.936,E2 13279.936} C_VEL
LIN {X 0,Y 330.474,Z 903.001,A -85,B 0,C 180,E1 13277.571,E2 13277.571} C_VEL
LIN {X 0,Y 322.333,Z 921.388,A -85,B 0,C 180,E1 13274.516,E2 13274.516} C_VEL
LIN {X 0,Y 315.456,Z 936.579,A -85,B 0,C 180,E1 13271.492,E2 13271.492} C_VEL
LIN {X 0,Y 308.712,Z 951.258,A -85,B 0,C 180,E1 13267.984,E2 13267.984} C_VEL
LIN {X 0,Y 302.766,Z 964.703,A -85,B 0,C 180,E1 13264.159,E2 13264.159} C_VEL
LIN {X 0,Y 297.93,Z 976.057,A -85,B 0,C 180,E1 13260.231,E2 13260.231} C_VEL
LIN {X 0,Y 293.874,Z 986.682,A -85,B 0,C 180,E1 13255.823,E2 13255.823} C_VEL
LIN {X 0,Y 291.246,Z 994.625,A -85,B 0,C 180,E1 13251.769,E2 13251.769} C_VEL
LIN {X 0,Y 289.328,Z 1001.995,A -85,B 0,C 180,E1 13247.088,E2 13247.088} C_VEL
LIN {X 0,Y 288.425,Z 1006.881,A -85,B 0,C 180,E1 13243.028,E2 13243.028} C_VEL
LIN {X 0,Y 288.039,Z 1010.776,A -85,B 0,C 180,E1 13238.59,E2 13238.59} C_VEL
LIN {X 0,Y 287.963,Z 1012.865,A -85,B 0,C 180,E1 13234.586,E2 13234.586} C_VEL
LIN {X 0,Y 287.969,Z 1013.702,A -85,B 0,C 180,E1 13231.001,E2 13231.001} C_VEL
LIN {X 0,Y 287.953,Z 1013.458,A -85,B 0,C 180,E1 13227.021,E2 13227.021} C_VEL
LIN {X 0,Y 287.967,Z 1011.798,A -85,B 0,C 180,E1 13223.026,E2 13223.026} C_VEL
LIN {X 0,Y 288.133,Z 1009.257,A -85,B 0,C 180,E1 13219.409,E2 13219.409} C_VEL
LIN {X 0,Y 288.785,Z 1004.73,A -85,B 0,C 180,E1 13214.956,E2 13214.956} C_VEL
LIN {X 0,Y 290.049,Z 998.986,A -85,B 0,C 180,E1 13210.825,E2 13210.825} C_VEL
LIN {X 0,Y 292.319,Z 991.303,A -85,B 0,C 180,E1 13206.417,E2 13206.417} C_VEL
LIN {X 0,Y 295.38,Z 982.496,A -85,B 0,C 180,E1 13202.379,E2 13202.379} C_VEL
LIN {X 0,Y 299.706,Z 971.514,A -85,B 0,C 180,E1 13198.198,E2 13198.198} C_VEL
LIN {X 0,Y 304.672,Z 959.665,A -85,B 0,C 180,E1 13194.475,E2 13194.475} C_VEL
LIN {X 0,Y 310.963,Z 945.238,A -85,B 0,C 180,E1 13190.706,E2 13190.706} C_VEL
LIN {X 0,Y 317.598,Z 930.146,A -85,B 0,C 180,E1 13187.411,E2 13187.411} C_VEL
LIN {X 0,Y 324.466,Z 914.045,A -85,B 0,C 180,E1 13184.5,E2 13184.5} C_VEL
LIN {X 0,Y 331.606,Z 896.824,A -85,B 0,C 180,E1 13181.872,E2 13181.872} C_VEL
LIN {X 0,Y 338.564,Z 878.713,A -85,B 0,C 180,E1 13179.586,E2 13179.586} C_VEL
LIN {X 0,Y 345.755,Z 858.653,A -85,B 0,C 180,E1 13177.469,E2 13177.469} C_VEL
LIN {X 0,Y 351.885,Z 839.742,A -85,B 0,C 180,E1 13175.826,E2 13175.826} C_VEL
LIN {X 0,Y 358.357,Z 817.198,A -85,B 0,C 180,E1 13174.228,E2 13174.228} C_VEL
LIN {X 0,Y 363.652,Z 795.902,A -85,B 0,C 180,E1 13173.02,E2 13173.02} C_VEL
LIN {X 0,Y 368.307,Z 773.058,A -85,B 0,C 180,E1 13172.016,E2 13172.016} C_VEL
LIN {X 0,Y 372.132,Z 749.827,A -85,B 0,C 180,E1 13171.251,E2 13171.251} C_VEL
LIN {X 0,Y 374.607,Z 726.767,A -85,B 0,C 180,E1 13170.688,E2 13170.688} C_VEL
LIN {X 0,Y 389.232,Z 518.022,A -85,B 0,C 180,E1 13166.485,E2 13166.485} C_VEL
LIN {X 0,Y 389.384,Z 515.185,A -85,B 0,C 180,E1 13166.414,E2 13166.414} C_VEL
LIN {X 0,Y 379.598,Z 499.13,A -85,B 0,C 180,E1 13163.025,E2 13163.025} C_VEL
LIN {X 0,Y 371.161,Z 486.481,A -85,B 0,C 180,E1 13159.718,E2 13159.718} C_VEL
LIN {X 0,Y 364.716,Z 477.74,A -85,B 0,C 180,E1 13156.893,E2 13156.893} C_VEL
LIN {X 0,Y 359.757,Z 471.524,A -85,B 0,C 180,E1 13154.485,E2 13154.485} C_VEL
LIN {X 0,Y 356.041,Z 466.747,A -85,B 0,C 180,E1 13152.487,E2 13152.487} C_VEL
LIN {X 0,Y 352.289,Z 462.011,A -85,B 0,C 180,E1 13150.258,E2 13150.258} C_VEL
LIN {X 0,Y 347.837,Z 456.769,A -85,B 0,C 180,E1 13147.265,E2 13147.265} C_VEL
LIN {X 0,Y 346.777,Z 455.339,A -85,B 0,C 180,E1 13146.456,E2 13146.456} C_VEL
LIN {X 0,Y 343.526,Z 451.968,A -85,B 0,C 180,E1 13143.838,E2 13143.838} C_VEL
LIN {X 0,Y 341.997,Z 449.411,A -85,B 0,C 180,E1 13142.345,E2 13142.345} C_VEL
LIN {X 0,Y 338.556,Z 446.413,A -85,B 0,C 180,E1 13138.645,E2 13138.645} C_VEL
LIN {X 0,Y 336.907,Z 443.188,A -85,B 0,C 180,E1 13136.085,E2 13136.085} C_VEL
LIN {X 0,Y 333.755,Z 441.141,A -85,B 0,C 180,E1 13128.596,E2 13128.596} C_VEL
LIN {X 0,Y 333.603,Z 441.051,A -85,B 0,C 180,E1 13123.636,E2 13123.636} C_VEL
LIN {X 0,Y 335.549,Z 442.554,A -85,B 0,C 180,E1 13117.393,E2 13117.393} C_VEL
LIN {X 0,Y 337.221,Z 443.589,A -85,B 0,C 180,E1 13114.631,E2 13114.631} C_VEL
LIN {X 0,Y 339.178,Z 447.166,A -85,B 0,C 180,E1 13111.799,E2 13111.799} C_VEL
LIN {X 0,Y 342.444,Z 449.945,A -85,B 0,C 180,E1 13108.479,E2 13108.479} C_VEL
LIN {X 0,Y 345.169,Z 453.959,A -85,B 0,C 180,E1 13106.008,E2 13106.008} C_VEL
LIN {X 0,Y 347.565,Z 456.26,A -85,B 0,C 180,E1 13104.206,E2 13104.206} C_VEL
LIN {X 0,Y 350.728,Z 460.403,A -85,B 0,C 180,E1 13101.991,E2 13101.991} C_VEL
LIN {X 0,Y 352.377,Z 462.16,A -85,B 0,C 180,E1 13100.955,E2 13100.955} C_VEL
LIN {X 0,Y 356.17,Z 466.836,A -85,B 0,C 180,E1 13098.722,E2 13098.722} C_VEL
LIN {X 0,Y 361.754,Z 474.051,A -85,B 0,C 180,E1 13095.796,E2 13095.796} C_VEL
LIN {X 0,Y 366.301,Z 480.012,A -85,B 0,C 180,E1 13093.668,E2 13093.668} C_VEL
LIN {X 0,Y 373.044,Z 488.865,A -85,B 0,C 180,E1 13090.835,E2 13090.835} C_VEL
LIN {X 0,Y 381.154,Z 500.357,A -85,B 0,C 180,E1 13087.79,E2 13087.79} C_VEL
LIN {X 0,Y 388.586,Z 511.372,A -85,B 0,C 180,E1 13085.282,E2 13085.282} C_VEL
LIN {X 0,Y 389.065,Z 512.525,A -85,B 0,C 180,E1 13085.112,E2 13085.112} C_VEL
LIN {X 0,Y 374.71,Z 715.37,A -85,B 0,C 180,E1 13081.024,E2 13081.024} C_VEL
LIN {X 0,Y 371.705,Z 740.091,A -85,B 0,C 180,E1 13080.349,E2 13080.349} C_VEL
LIN {X 0,Y 368.069,Z 762.141,A -85,B 0,C 180,E1 13079.523,E2 13079.523} C_VEL
LIN {X 0,Y 363.328,Z 784.459,A -85,B 0,C 180,E1 13078.423,E2 13078.423} C_VEL
LIN {X 0,Y 357.893,Z 806.187,A -85,B 0,C 180,E1 13077.083,E2 13077.083} C_VEL
LIN {X 0,Y 352.057,Z 825.994,A -85,B 0,C 180,E1 13075.568,E2 13075.568} C_VEL
LIN {X 0,Y 344.946,Z 847.436,A -85,B 0,C 180,E1 13073.572,E2 13073.572} C_VEL
LIN {X 0,Y 338.227,Z 865.81,A -85,B 0,C 180,E1 13071.498,E2 13071.498} C_VEL
LIN {X 0,Y 331.004,Z 883.914,A -85,B 0,C 180,E1 13069.034,E2 13069.034} C_VEL
LIN {X 0,Y 324.154,Z 900.197,A -85,B 0,C 180,E1 13066.404,E2 13066.404} C_VEL
LIN {X 0,Y 317.414,Z 915.256,A -85,B 0,C 180,E1 13063.474,E2 13063.474} C_VEL
LIN {X 0,Y 310.965,Z 929.587,A -85,B 0,C 180,E1 13060.18,E2 13060.18} C_VEL
LIN {X 0,Y 305.04,Z 942.49,A -85,B 0,C 180,E1 13056.582,E2 13056.582} C_VEL
LIN {X 0,Y 299.654,Z 954.683,A -85,B 0,C 180,E1 13052.48,E2 13052.48} C_VEL
LIN {X 0,Y 295.728,Z 964.082,A -85,B 0,C 180,E1 13048.638,E2 13048.638} C_VEL
LIN {X 0,Y 292.333,Z 973.083,A -85,B 0,C 180,E1 13044.105,E2 13044.105} C_VEL
LIN {X 0,Y 290.205,Z 979.793,A -85,B 0,C 180,E1 13039.874,E2 13039.874} C_VEL
LIN {X 0,Y 288.855,Z 985.196,A -85,B 0,C 180,E1 13035.358,E2 13035.358} C_VEL
LIN {X 0,Y 288.247,Z 988.789,A -85,B 0,C 180,E1 13031.26,E2 13031.26} C_VEL
LIN {X 0,Y 288.06,Z 990.576,A -85,B 0,C 180,E1 13028.287,E2 13028.287} C_VEL
LIN {X 0,Y 287.009,Z 991.37,A -85,B 0,C 180,E1 13026.764,E2 13026.764} C_VEL
LIN {X 0,Y 282.879,Z 992.281,A -85,B 0,C 180,E1 13024.195,E2 13024.195} C_VEL
LIN {X 0,Y 280.258,Z 992.516,A -85,B 0,C 180,E1 13022.087,E2 13022.087} C_VEL
LIN {X 0,Y 279.994,Z 992.474,A -85,B 0,C 180,E1 13021.286,E2 13021.286} C_VEL
LIN {X 0,Y 280.02,Z 991.795,A -85,B 0,C 180,E1 13017.367,E2 13017.367} C_VEL
LIN {X 0,Y 280.215,Z 990.076,A -85,B 0,C 180,E1 13013.404,E2 13013.404} C_VEL
LIN {X 0,Y 280.893,Z 986.544,A -85,B 0,C 180,E1 13008.684,E2 13008.684} C_VEL
LIN {X 0,Y 282.089,Z 982.162,A -85,B 0,C 180,E1 13004.56,E2 13004.56} C_VEL
LIN {X 0,Y 284.54,Z 975.285,A -85,B 0,C 180,E1 12999.679,E2 12999.679} C_VEL
LIN {X 0,Y 287.72,Z 967.764,A -85,B 0,C 180,E1 12995.476,E2 12995.476} C_VEL
LIN {X 0,Y 292.261,Z 958.039,A -85,B 0,C 180,E1 12991.105,E2 12991.105} C_VEL
LIN {X 0,Y 297.938,Z 946.769,A -85,B 0,C 180,E1 12986.94,E2 12986.94} C_VEL
LIN {X 0,Y 304.449,Z 934.031,A -85,B 0,C 180,E1 12983.128,E2 12983.128} C_VEL
LIN {X 0,Y 312.043,Z 919.269,A -85,B 0,C 180,E1 12979.466,E2 12979.466} C_VEL
LIN {X 0,Y 319.392,Z 904.665,A -85,B 0,C 180,E1 12976.471,E2 12976.471} C_VEL
LIN {X 0,Y 327.489,Z 887.811,A -85,B 0,C 180,E1 12973.598,E2 12973.598} C_VEL
LIN {X 0,Y 335.558,Z 870.1,A -85,B 0,C 180,E1 12971.081,E2 12971.081} C_VEL
LIN {X 0,Y 343.391,Z 851.143,A -85,B 0,C 180,E1 12968.878,E2 12968.878} C_VEL
LIN {X 0,Y 350.973,Z 831.174,A -85,B 0,C 180,E1 12966.955,E2 12966.955} C_VEL
LIN {X 0,Y 357.556,Z 811.491,A -85,B 0,C 180,E1 12965.405,E2 12965.405} C_VEL
LIN {X 0,Y 364.07,Z 789.152,A -85,B 0,C 180,E1 12963.979,E2 12963.979} C_VEL
LIN {X 0,Y 369.241,Z 768.073,A -85,B 0,C 180,E1 12962.907,E2 12962.907} C_VEL
LIN {X 0,Y 373.687,Z 745.285,A -85,B 0,C 180,E1 12962.015,E2 12962.015} C_VEL
LIN {X 0,Y 377.165,Z 722.046,A -85,B 0,C 180,E1 12961.345,E2 12961.345} C_VEL
LIN {X 0,Y 395.57,Z 520.925,A -85,B 0,C 180,E1 12957.171,E2 12957.171} C_VEL
LIN {X 0,Y 392.213,Z 514.409,A -85,B 0,C 180,E1 12955.028,E2 12955.028} C_VEL
LIN {X 0,Y 389.32,Z 508.855,A -85,B 0,C 180,E1 12952.623,E2 12952.623} C_VEL
LIN {X 0,Y 387.346,Z 504.986,A -85,B 0,C 180,E1 12950.192,E2 12950.192} C_VEL
LIN {X 0,Y 386.109,Z 502.693,A -85,B 0,C 180,E1 12946.218,E2 12946.218} C_VEL
LIN {X 0,Y 387.341,Z 504.985,A -85,B 0,C 180,E1 12942.267,E2 12942.267} C_VEL
LIN {X 0,Y 387.945,Z 506.349,A -85,B 0,C 180,E1 12941.363,E2 12941.363} C_VEL
LIN {X 0,Y 389.954,Z 510.164,A -85,B 0,C 180,E1 12939.2,E2 12939.2} C_VEL
LIN {X 0,Y 392.208,Z 514.594,A -85,B 0,C 180,E1 12937.4,E2 12937.4} C_VEL
LIN {X 0,Y 395.548,Z 522.365,A -85,B 0,C 180,E1 12935.191,E2 12935.191} C_VEL
LIN {X 0,Y 378.394,Z 712.65,A -85,B 0,C 180,E1 12931.257,E2 12931.257} C_VEL
LIN {X 0,Y 375.458,Z 739.732,A -85,B 0,C 180,E1 12930.638,E2 12930.638} C_VEL
LIN {X 0,Y 371.574,Z 763.161,A -85,B 0,C 180,E1 12929.951,E2 12929.951} C_VEL
LIN {X 0,Y 366.953,Z 784.083,A -85,B 0,C 180,E1 12929.131,E2 12929.131} C_VEL
LIN {X 0,Y 361.277,Z 806.1,A -85,B 0,C 180,E1 12928.028,E2 12928.028} C_VEL
LIN {X 0,Y 355.113,Z 826.2,A -85,B 0,C 180,E1 12926.75,E2 12926.75} C_VEL
LIN {X 0,Y 348.023,Z 847.041,A -85,B 0,C 180,E1 12925.131,E2 12925.131} C_VEL
LIN {X 0,Y 340.871,Z 865.715,A -85,B 0,C 180,E1 12923.35,E2 12923.35} C_VEL
LIN {X 0,Y 332.795,Z 885.368,A -85,B 0,C 180,E1 12921.097,E2 12921.097} C_VEL
LIN {X 0,Y 324.995,Z 902.943,A -85,B 0,C 180,E1 12918.654,E2 12918.654} C_VEL
LIN {X 0,Y 316.452,Z 921.295,A -85,B 0,C 180,E1 12915.572,E2 12915.572} C_VEL
LIN {X 0,Y 308.858,Z 937.307,A -85,B 0,C 180,E1 12912.332,E2 12912.332} C_VEL
LIN {X 0,Y 301.811,Z 951.783,A -85,B 0,C 180,E1 12908.771,E2 12908.771} C_VEL
LIN {X 0,Y 295.579,Z 965.057,A -85,B 0,C 180,E1 12904.873,E2 12904.873} C_VEL
LIN {X 0,Y 290.496,Z 976.341,A -85,B 0,C 180,E1 12900.859,E2 12900.859} C_VEL
LIN {X 0,Y 286.052,Z 987.248,A -85,B 0,C 180,E1 12896.136,E2 12896.136} C_VEL
LIN {X 0,Y 283.245,Z 995.358,A -85,B 0,C 180,E1 12891.816,E2 12891.816} C_VEL
LIN {X 0,Y 281.339,Z 1002.237,A -85,B 0,C 180,E1 12887.162,E2 12887.162} C_VEL
LIN {X 0,Y 280.414,Z 1007.026,A -85,B 0,C 180,E1 12882.987,E2 12882.987} C_VEL
LIN {X 0,Y 280.026,Z 1010.846,A -85,B 0,C 180,E1 12878.217,E2 12878.217} C_VEL
LIN {X 0,Y 279.966,Z 1012.643,A -85,B 0,C 180,E1 12874.512,E2 12874.512} C_VEL
LIN {X 0,Y 279.971,Z 1013.459,A -85,B 0,C 180,E1 12870.597,E2 12870.597} C_VEL
LIN {X 0,Y 279.959,Z 1013.013,A -85,B 0,C 180,E1 12866.526,E2 12866.526} C_VEL
LIN {X 0,Y 279.97,Z 1011.485,A -85,B 0,C 180,E1 12862.826,E2 12862.826} C_VEL
LIN {X 0,Y 280.163,Z 1008.936,A -85,B 0,C 180,E1 12859.104,E2 12859.104} C_VEL
LIN {X 0,Y 280.875,Z 1004.388,A -85,B 0,C 180,E1 12854.522,E2 12854.522} C_VEL
LIN {X 0,Y 282.23,Z 998.725,A -85,B 0,C 180,E1 12850.34,E2 12850.34} C_VEL
LIN {X 0,Y 284.698,Z 990.915,A -85,B 0,C 180,E1 12845.746,E2 12845.746} C_VEL
LIN {X 0,Y 287.983,Z 982.093,A -85,B 0,C 180,E1 12841.606,E2 12841.606} C_VEL
LIN {X 0,Y 292.848,Z 970.47,A -85,B 0,C 180,E1 12837.129,E2 12837.129} C_VEL
LIN {X 0,Y 298.137,Z 958.588,A -85,B 0,C 180,E1 12833.357,E2 12833.357} C_VEL
LIN {X 0,Y 304.487,Z 944.711,A -85,B 0,C 180,E1 12829.701,E2 12829.701} C_VEL
LIN {X 0,Y 311.455,Z 929.572,A -85,B 0,C 180,E1 12826.363,E2 12826.363} C_VEL
LIN {X 0,Y 318.709,Z 913.221,A -85,B 0,C 180,E1 12823.396,E2 12823.396} C_VEL
LIN {X 0,Y 326.316,Z 895.461,A -85,B 0,C 180,E1 12820.691,E2 12820.691} C_VEL
LIN {X 0,Y 333.299,Z 877.926,A -85,B 0,C 180,E1 12818.478,E2 12818.478} C_VEL
LIN {X 0,Y 341.034,Z 856.881,A -85,B 0,C 180,E1 12816.28,E2 12816.28} C_VEL
LIN {X 0,Y 347.458,Z 837.567,A -85,B 0,C 180,E1 12814.625,E2 12814.625} C_VEL
LIN {X 0,Y 353.853,Z 815.665,A -85,B 0,C 180,E1 12813.104,E2 12813.104} C_VEL
LIN {X 0,Y 359.4,Z 793.86,A -85,B 0,C 180,E1 12811.887,E2 12811.887} C_VEL
LIN {X 0,Y 364.026,Z 771.358,A -85,B 0,C 180,E1 12810.923,E2 12810.923} C_VEL
LIN {X 0,Y 367.994,Z 747.041,A -85,B 0,C 180,E1 12810.149,E2 12810.149} C_VEL
LIN {X 0,Y 370.405,Z 724.391,A -85,B 0,C 180,E1 12809.605,E2 12809.605} C_VEL
LIN {X 0,Y 385.187,Z 519.723,A -85,B 0,C 180,E1 12805.483,E2 12805.483} C_VEL
LIN {X 0,Y 376.617,Z 505.399,A -85,B 0,C 180,E1 12802.393,E2 12802.393} C_VEL
LIN {X 0,Y 368.757,Z 493.46,A -85,B 0,C 180,E1 12799.234,E2 12799.234} C_VEL
LIN {X 0,Y 362.482,Z 484.883,A -85,B 0,C 180,E1 12796.423,E2 12796.423} C_VEL
LIN {X 0,Y 357.764,Z 478.85,A -85,B 0,C 180,E1 12794.071,E2 12794.071} C_VEL
LIN {X 0,Y 354.129,Z 474.128,A -85,B 0,C 180,E1 12792.059,E2 12792.059} C_VEL
LIN {X 0,Y 349.772,Z 468.626,A -85,B 0,C 180,E1 12789.377,E2 12789.377} C_VEL
LIN {X 0,Y 346.204,Z 464.25,A -85,B 0,C 180,E1 12786.883,E2 12786.883} C_VEL
LIN {X 0,Y 345.239,Z 463.021,A -85,B 0,C 180,E1 12786.151,E2 12786.151} C_VEL
LIN {X 0,Y 341.961,Z 459.456,A -85,B 0,C 180,E1 12783.436,E2 12783.436} C_VEL
LIN {X 0,Y 340.732,Z 457.264,A -85,B 0,C 180,E1 12782.186,E2 12782.186} C_VEL
LIN {X 0,Y 337.316,Z 454.254,A -85,B 0,C 180,E1 12778.471,E2 12778.471} C_VEL
LIN {X 0,Y 335.698,Z 451.062,A -85,B 0,C 180,E1 12775.9,E2 12775.9} C_VEL
LIN {X 0,Y 332.644,Z 449.033,A -85,B 0,C 180,E1 12768.381,E2 12768.381} C_VEL
LIN {X 0,Y 332.56,Z 449.005,A -85,B 0,C 180,E1 12763.403,E2 12763.403} C_VEL
LIN {X 0,Y 334.897,Z 450.697,A -85,B 0,C 180,E1 12756.603,E2 12756.603} C_VEL
LIN {X 0,Y 336.011,Z 451.455,A -85,B 0,C 180,E1 12754.816,E2 12754.816} C_VEL
LIN {X 0,Y 337.964,Z 455.034,A -85,B 0,C 180,E1 12751.939,E2 12751.939} C_VEL
LIN {X 0,Y 341.05,Z 457.71,A -85,B 0,C 180,E1 12748.74,E2 12748.74} C_VEL
LIN {X 0,Y 343.859,Z 461.807,A -85,B 0,C 180,E1 12746.162,E2 12746.162} C_VEL
LIN {X 0,Y 346.048,Z 463.953,A -85,B 0,C 180,E1 12744.495,E2 12744.495} C_VEL
LIN {X 0,Y 349.321,Z 468.208,A -85,B 0,C 180,E1 12742.174,E2 12742.174} C_VEL
LIN {X 0,Y 350.865,Z 470.012,A -85,B 0,C 180,E1 12741.175,E2 12741.175} C_VEL
LIN {X 0,Y 355.551,Z 475.933,A -85,B 0,C 180,E1 12738.41,E2 12738.41} C_VEL
LIN {X 0,Y 359.991,Z 481.721,A -85,B 0,C 180,E1 12736.078,E2 12736.078} C_VEL
LIN {X 0,Y 364.484,Z 487.684,A -85,B 0,C 180,E1 12733.941,E2 12733.941} C_VEL
LIN {X 0,Y 370.959,Z 496.349,A -85,B 0,C 180,E1 12731.171,E2 12731.171} C_VEL
LIN {X 0,Y 379.991,Z 509.246,A -85,B 0,C 180,E1 12727.748,E2 12727.748} C_VEL
LIN {X 0,Y 384.836,Z 516.855,A -85,B 0,C 180,E1 12726.064,E2 12726.064} C_VEL
LIN {X 0,Y 370.233,Z 716.493,A -85,B 0,C 180,E1 12722.032,E2 12722.032} C_VEL
LIN {X 0,Y 367.152,Z 740.782,A -85,B 0,C 180,E1 12721.364,E2 12721.364} C_VEL
LIN {X 0,Y 363.365,Z 763.031,A -85,B 0,C 180,E1 12720.527,E2 12720.527} C_VEL
LIN {X 0,Y 358.66,Z 784.477,A -85,B 0,C 180,E1 12719.468,E2 12719.468} C_VEL
LIN {X 0,Y 353.342,Z 805.32,A -85,B 0,C 180,E1 12718.194,E2 12718.194} C_VEL
LIN {X 0,Y 347.035,Z 826.141,A -85,B 0,C 180,E1 12716.61,E2 12716.61} C_VEL
LIN {X 0,Y 339.947,Z 846.967,A -85,B 0,C 180,E1 12714.68,E2 12714.68} C_VEL
LIN {X 0,Y 333.206,Z 864.821,A -85,B 0,C 180,E1 12712.674,E2 12712.674} C_VEL
LIN {X 0,Y 325.452,Z 883.672,A -85,B 0,C 180,E1 12710.12,E2 12710.12} C_VEL
LIN {X 0,Y 318.484,Z 899.628,A -85,B 0,C 180,E1 12707.534,E2 12707.534} C_VEL
LIN {X 0,Y 311.276,Z 915.192,A -85,B 0,C 180,E1 12704.503,E2 12704.503} C_VEL
LIN {X 0,Y 304.497,Z 929.596,A -85,B 0,C 180,E1 12701.165,E2 12701.165} C_VEL
LIN {X 0,Y 298.261,Z 942.53,A -85,B 0,C 180,E1 12697.506,E2 12697.506} C_VEL
LIN {X 0,Y 292.795,Z 954.295,A -85,B 0,C 180,E1 12693.518,E2 12693.518} C_VEL
LIN {X 0,Y 288.543,Z 963.78,A -85,B 0,C 180,E1 12689.597,E2 12689.597} C_VEL
LIN {X 0,Y 284.865,Z 972.908,A -85,B 0,C 180,E1 12684.96,E2 12684.96} C_VEL
LIN {X 0,Y 282.603,Z 979.431,A -85,B 0,C 180,E1 12680.796,E2 12680.796} C_VEL
LIN {X 0,Y 281.002,Z 985.212,A -85,B 0,C 180,E1 12675.992,E2 12675.992} C_VEL
LIN {X 0,Y 280.336,Z 988.762,A -85,B 0,C 180,E1 12671.917,E2 12671.917} C_VEL
LIN {X 0,Y 280.048,Z 991.285,A -85,B 0,C 180,E1 12667.535,E2 12667.535} C_VEL
LIN {X 0,Y 279.976,Z 992.333,A -85,B 0,C 180,E1 12663.481,E2 12663.481} C_VEL
LIN {X 0,Y 279.994,Z 992.474,A -85,B 0,C 180,E1 12661.286,E2 12661.286} C_VEL
LIN {X 0,Y 279.138,Z 992.38,A -85,B 0,C 180,E1 12659.821,E2 12659.821} C_VEL
LIN {X 0,Y 275.678,Z 992.039,A -85,B 0,C 180,E1 12657.502,E2 12657.502} C_VEL
LIN {X 0,Y 272.56,Z 991.371,A -85,B 0,C 180,E1 12655.122,E2 12655.122} C_VEL
LIN {X 0,Y 272.185,Z 990.862,A -85,B 0,C 180,E1 12654.068,E2 12654.068} C_VEL
LIN {X 0,Y 272.74,Z 987.986,A -85,B 0,C 180,E1 12649.536,E2 12649.536} C_VEL
LIN {X 0,Y 273.976,Z 983.517,A -85,B 0,C 180,E1 12644.922,E2 12644.922} C_VEL
LIN {X 0,Y 276.087,Z 977.786,A -85,B 0,C 180,E1 12640.411,E2 12640.411} C_VEL
LIN {X 0,Y 279.377,Z 970.196,A -85,B 0,C 180,E1 12635.807,E2 12635.807} C_VEL
LIN {X 0,Y 283.792,Z 961.301,A -85,B 0,C 180,E1 12631.43,E2 12631.43} C_VEL
LIN {X 0,Y 289.49,Z 950.373,A -85,B 0,C 180,E1 12627.124,E2 12627.124} C_VEL
LIN {X 0,Y 296.354,Z 937.765,A -85,B 0,C 180,E1 12623.041,E2 12623.041} C_VEL
LIN {X 0,Y 303.484,Z 924.644,A -85,B 0,C 180,E1 12619.555,E2 12619.555} C_VEL
LIN {X 0,Y 311.89,Z 908.83,A -85,B 0,C 180,E1 12616.09,E2 12616.09} C_VEL
LIN {X 0,Y 320.34,Z 892.415,A -85,B 0,C 180,E1 12613.123,E2 12613.123} C_VEL
LIN {X 0,Y 328.547,Z 875.174,A -85,B 0,C 180,E1 12610.57,E2 12610.57} C_VEL
LIN {X 0,Y 337.184,Z 855.746,A -85,B 0,C 180,E1 12608.184,E2 12608.184} C_VEL
LIN {X 0,Y 344.582,Z 837.37,A -85,B 0,C 180,E1 12606.331,E2 12606.331} C_VEL
LIN {X 0,Y 352.282,Z 815.935,A -85,B 0,C 180,E1 12604.559,E2 12604.559} C_VEL
LIN {X 0,Y 359.092,Z 794.277,A -85,B 0,C 180,E1 12603.113,E2 12603.113} C_VEL
LIN {X 0,Y 364.766,Z 772.438,A -85,B 0,C 180,E1 12601.964,E2 12601.964} C_VEL
LIN {X 0,Y 369.736,Z 749.007,A -85,B 0,C 180,E1 12601.008,E2 12601.008} C_VEL
LIN {X 0,Y 373.3,Z 726.996,A -85,B 0,C 180,E1 12600.344,E2 12600.344} C_VEL
LIN {X 0,Y 376.672,Z 694.678,A -85,B 0,C 180,E1 12599.63,E2 12599.63} C_VEL
LIN {X 0,Y 392.677,Z 526.17,A -85,B 0,C 180,E1 12596.15,E2 12596.15} C_VEL
LIN {X 0,Y 389.659,Z 520.006,A -85,B 0,C 180,E1 12593.962,E2 12593.962} C_VEL
LIN {X 0,Y 387.796,Z 516.329,A -85,B 0,C 180,E1 12592.221,E2 12592.221} C_VEL
LIN {X 0,Y 386.13,Z 512.82,A -85,B 0,C 180,E1 12590.01,E2 12590.01} C_VEL
LIN {X 0,Y 385.02,Z 510.628,A -85,B 0,C 180,E1 12586.178,E2 12586.178} C_VEL
LIN {X 0,Y 386.324,Z 513.063,A -85,B 0,C 180,E1 12582.141,E2 12582.141} C_VEL
LIN {X 0,Y 388.562,Z 517.921,A -85,B 0,C 180,E1 12579.437,E2 12579.437} C_VEL
LIN {X 0,Y 390.508,Z 522.018,A -85,B 0,C 180,E1 12577.772,E2 12577.772} C_VEL
LIN {X 0,Y 392.657,Z 527.579,A -85,B 0,C 180,E1 12576.199,E2 12576.199} C_VEL
LIN {X 0,Y 373.26,Z 731.949,A -85,B 0,C 180,E1 12571.958,E2 12571.958} C_VEL
LIN {X 0,Y 369.477,Z 755.75,A -85,B 0,C 180,E1 12571.314,E2 12571.314} C_VEL
LIN {X 0,Y 364.365,Z 779.869,A -85,B 0,C 180,E1 12570.451,E2 12570.451} C_VEL
LIN {X 0,Y 358.816,Z 801.121,A -85,B 0,C 180,E1 12569.44,E2 12569.44} C_VEL
LIN {X 0,Y 351.767,Z 823.977,A -85,B 0,C 180,E1 12568.049,E2 12568.049} C_VEL
LIN {X 0,Y 344.378,Z 845.159,A -85,B 0,C 180,E1 12566.442,E2 12566.442} C_VEL
LIN {X 0,Y 336.381,Z 865.315,A -85,B 0,C 180,E1 12564.537,E2 12564.537} C_VEL
LIN {X 0,Y 327.988,Z 884.91,A -85,B 0,C 180,E1 12562.29,E2 12562.29} C_VEL
LIN {X 0,Y 320.135,Z 901.896,A -85,B 0,C 180,E1 12559.93,E2 12559.93} C_VEL
LIN {X 0,Y 311.168,Z 920.315,A -85,B 0,C 180,E1 12556.842,E2 12556.842} C_VEL
LIN {X 0,Y 303.154,Z 936.343,A -85,B 0,C 180,E1 12553.582,E2 12553.582} C_VEL
LIN {X 0,Y 295.7,Z 950.904,A -85,B 0,C 180,E1 12549.981,E2 12549.981} C_VEL
LIN {X 0,Y 289.047,Z 964.256,A -85,B 0,C 180,E1 12546.025,E2 12546.025} C_VEL
LIN {X 0,Y 283.581,Z 975.572,A -85,B 0,C 180,E1 12541.935,E2 12541.935} C_VEL
LIN {X 0,Y 278.756,Z 986.568,A -85,B 0,C 180,E1 12537.105,E2 12537.105} C_VEL
LIN {X 0,Y 275.758,Z 994.44,A -85,B 0,C 180,E1 12532.834,E2 12532.834} C_VEL
LIN {X 0,Y 273.552,Z 1001.686,A -85,B 0,C 180,E1 12527.886,E2 12527.886} C_VEL
LIN {X 0,Y 272.493,Z 1006.603,A -85,B 0,C 180,E1 12523.505,E2 12523.505} C_VEL
LIN {X 0,Y 272.043,Z 1010.449,A -85,B 0,C 180,E1 12518.637,E2 12518.637} C_VEL
LIN {X 0,Y 271.969,Z 1012.272,A -85,B 0,C 180,E1 12514.857,E2 12514.857} C_VEL
LIN {X 0,Y 271.981,Z 1013.105,A -85,B 0,C 180,E1 12511.06,E2 12511.06} C_VEL
LIN {X 0,Y 271.962,Z 1012.841,A -85,B 0,C 180,E1 12506.845,E2 12506.845} C_VEL
LIN {X 0,Y 271.973,Z 1011.284,A -85,B 0,C 180,E1 12502.826,E2 12502.826} C_VEL
LIN {X 0,Y 272.173,Z 1008.773,A -85,B 0,C 180,E1 12498.994,E2 12498.994} C_VEL
LIN {X 0,Y 272.873,Z 1004.563,A -85,B 0,C 180,E1 12494.493,E2 12494.493} C_VEL
LIN {X 0,Y 274.362,Z 998.677,A -85,B 0,C 180,E1 12489.974,E2 12489.974} C_VEL
LIN {X 0,Y 276.827,Z 991.351,A -85,B 0,C 180,E1 12485.466,E2 12485.466} C_VEL
LIN {X 0,Y 280.433,Z 982.143,A -85,B 0,C 180,E1 12481.003,E2 12481.003} C_VEL
LIN {X 0,Y 285.292,Z 971.194,A -85,B 0,C 180,E1 12476.626,E2 12476.626} C_VEL
LIN {X 0,Y 290.779,Z 959.413,A -85,B 0,C 180,E1 12472.767,E2 12472.767} C_VEL
LIN {X 0,Y 297.937,Z 944.505,A -85,B 0,C 180,E1 12468.739,E2 12468.739} C_VEL
LIN {X 0,Y 304.987,Z 929.845,A -85,B 0,C 180,E1 12465.457,E2 12465.457} C_VEL
LIN {X 0,Y 312.508,Z 913.631,A -85,B 0,C 180,E1 12462.46,E2 12462.46} C_VEL
LIN {X 0,Y 320.143,Z 896.554,A -85,B 0,C 180,E1 12459.809,E2 12459.809} C_VEL
LIN {X 0,Y 327.883,Z 877.749,A -85,B 0,C 180,E1 12457.415,E2 12457.415} C_VEL
LIN {X 0,Y 335.882,Z 856.727,A -85,B 0,C 180,E1 12455.213,E2 12455.213} C_VEL
LIN {X 0,Y 342.506,Z 837.431,A -85,B 0,C 180,E1 12453.558,E2 12453.558} C_VEL
LIN {X 0,Y 349.09,Z 815.549,A -85,B 0,C 180,E1 12452.04,E2 12452.04} C_VEL
LIN {X 0,Y 354.789,Z 793.734,A -85,B 0,C 180,E1 12450.827,E2 12450.827} C_VEL
LIN {X 0,Y 359.519,Z 771.315,A -85,B 0,C 180,E1 12449.871,E2 12449.871} C_VEL
LIN {X 0,Y 363.552,Z 747.312,A -85,B 0,C 180,E1 12449.107,E2 12449.107} C_VEL
LIN {X 0,Y 366.036,Z 724.747,A -85,B 0,C 180,E1 12448.563,E2 12448.563} C_VEL
LIN {X 0,Y 381.057,Z 524.058,A -85,B 0,C 180,E1 12444.513,E2 12444.513} C_VEL
LIN {X 0,Y 372.822,Z 510.359,A -85,B 0,C 180,E1 12441.432,E2 12441.432} C_VEL
LIN {X 0,Y 366.107,Z 500.084,A -85,B 0,C 180,E1 12438.634,E2 12438.634} C_VEL
LIN {X 0,Y 360.12,Z 491.836,A -85,B 0,C 180,E1 12435.871,E2 12435.871} C_VEL
LIN {X 0,Y 355.787,Z 486.171,A -85,B 0,C 180,E1 12433.654,E2 12433.654} C_VEL
LIN {X 0,Y 352.347,Z 481.633,A -85,B 0,C 180,E1 12431.706,E2 12431.706} C_VEL
LIN {X 0,Y 348.047,Z 476.158,A -85,B 0,C 180,E1 12429.007,E2 12429.007} C_VEL
LIN {X 0,Y 344.557,Z 471.726,A -85,B 0,C 180,E1 12426.498,E2 12426.498} C_VEL
LIN {X 0,Y 343.063,Z 470.171,A -85,B 0,C 180,E1 12425.351,E2 12425.351} C_VEL
LIN {X 0,Y 340.083,Z 466.347,A -85,B 0,C 180,E1 12422.696,E2 12422.696} C_VEL
LIN {X 0,Y 339.293,Z 465.021,A -85,B 0,C 180,E1 12421.857,E2 12421.857} C_VEL
LIN {X 0,Y 335.828,Z 461.706,A -85,B 0,C 180,E1 12417.952,E2 12417.952} C_VEL
LIN {X 0,Y 334.601,Z 458.989,A -85,B 0,C 180,E1 12415.887,E2 12415.887} C_VEL
LIN {X 0,Y 331.557,Z 456.956,A -85,B 0,C 180,E1 12408.343,E2 12408.343} C_VEL
LIN {X 0,Y 331.457,Z 456.923,A -85,B 0,C 180,E1 12403.527,E2 12403.527} C_VEL
LIN {X 0,Y 333.633,Z 458.545,A -85,B 0,C 180,E1 12396.913,E2 12396.913} C_VEL
LIN {X 0,Y 334.804,Z 459.319,A -85,B 0,C 180,E1 12395.002,E2 12395.002} C_VEL
LIN {X 0,Y 336.794,Z 462.955,A -85,B 0,C 180,E1 12392.026,E2 12392.026} C_VEL
LIN {X 0,Y 339.672,Z 465.488,A -85,B 0,C 180,E1 12388.993,E2 12388.993} C_VEL
LIN {X 0,Y 342.552,Z 469.655,A -85,B 0,C 180,E1 12386.317,E2 12386.317} C_VEL
LIN {X 0,Y 344.496,Z 471.566,A -85,B 0,C 180,E1 12384.821,E2 12384.821} C_VEL
LIN {X 0,Y 347.91,Z 476.011,A -85,B 0,C 180,E1 12382.359,E2 12382.359} C_VEL
LIN {X 0,Y 349.479,Z 478.036,A -85,B 0,C 180,E1 12381.318,E2 12381.318} C_VEL
LIN {X 0,Y 353.811,Z 483.518,A -85,B 0,C 180,E1 12378.729,E2 12378.729} C_VEL
LIN {X 0,Y 358.153,Z 489.265,A -85,B 0,C 180,E1 12376.405,E2 12376.405} C_VEL
LIN {X 0,Y 362.777,Z 495.487,A -85,B 0,C 180,E1 12374.169,E2 12374.169} C_VEL
LIN {X 0,Y 369.975,Z 505.379,A -85,B 0,C 180,E1 12371.061,E2 12371.061} C_VEL
LIN {X 0,Y 378.248,Z 517.511,A -85,B 0,C 180,E1 12367.902,E2 12367.902} C_VEL
LIN {X 0,Y 380.689,Z 521.443,A -85,B 0,C 180,E1 12367.032,E2 12367.032} C_VEL
LIN {X 0,Y 365.873,Z 717.145,A -85,B 0,C 180,E1 12363.072,E2 12363.072} C_VEL
LIN {X 0,Y 362.725,Z 741.2,A -85,B 0,C 180,E1 12362.409,E2 12362.409} C_VEL
LIN {X 0,Y 358.868,Z 763.296,A -85,B 0,C 180,E1 12361.58,E2 12361.58} C_VEL
LIN {X 0,Y 353.815,Z 785.67,A -85,B 0,C 180,E1 12360.474,E2 12360.474} C_VEL
LIN {X 0,Y 348.046,Z 807.309,A -85,B 0,C 180,E1 12359.132,E2 12359.132} C_VEL
LIN {X 0,Y 341.852,Z 827.108,A -85,B 0,C 180,E1 12357.612,E2 12357.612} C_VEL
LIN {X 0,Y 334.27,Z 848.523,A -85,B 0,C 180,E1 12355.602,E2 12355.602} C_VEL
LIN {X 0,Y 326.838,Z 867.549,A -85,B 0,C 180,E1 12353.427,E2 12353.427} C_VEL
LIN {X 0,Y 319.09,Z 885.523,A -85,B 0,C 180,E1 12350.923,E2 12350.923} C_VEL
LIN {X 0,Y 311.368,Z 902.43,A -85,B 0,C 180,E1 12348.099,E2 12348.099} C_VEL
LIN {X 0,Y 304.052,Z 917.509,A -85,B 0,C 180,E1 12345.051,E2 12345.051} C_VEL
LIN {X 0,Y 296.389,Z 932.941,A -85,B 0,C 180,E1 12341.277,E2 12341.277} C_VEL
LIN {X 0,Y 290.37,Z 945.012,A -85,B 0,C 180,E1 12337.711,E2 12337.711} C_VEL
LIN {X 0,Y 284.783,Z 956.374,A -85,B 0,C 180,E1 12333.617,E2 12333.617} C_VEL
LIN {X 0,Y 280.303,Z 966.123,A -85,B 0,C 180,E1 12329.381,E2 12329.381} C_VEL
LIN {X 0,Y 276.754,Z 974.464,A -85,B 0,C 180,E1 12324.812,E2 12324.812} C_VEL
LIN {X 0,Y 274.321,Z 981.302,A -85,B 0,C 180,E1 12320.13,E2 12320.13} C_VEL
LIN {X 0,Y 272.968,Z 986.056,A -85,B 0,C 180,E1 12315.788,E2 12315.788} C_VEL
LIN {X 0,Y 272.276,Z 989.676,A -85,B 0,C 180,E1 12311.342,E2 12311.342} C_VEL
LIN {X 0,Y 272.022,Z 991.849,A -85,B 0,C 180,E1 12306.834,E2 12306.834} C_VEL
LIN {X 0,Y 271.985,Z 992.676,A -85,B 0,C 180,E1 12303.111,E2 12303.111} C_VEL
LIN {X 0,Y 272.024,Z 992.554,A -85,B 0,C 180,E1 12298.778,E2 12298.778} C_VEL
LIN {X 0,Y 272.174,Z 990.956,A -85,B 0,C 180,E1 12294.254,E2 12294.254} C_VEL
LIN {X 0,Y 272.185,Z 990.862,A -85,B 0,C 180,E1 12294.068,E2 12294.068} C_VEL
LIN {X 0,Y 271.328,Z 990.11,A -85,B 0,C 180,E1 12292.452,E2 12292.452} C_VEL
LIN {X 0,Y 265.707,Z 987.298,A -85,B 0,C 180,E1 12287.979,E2 12287.979} C_VEL
LIN {X 0,Y 265.428,Z 986.171,A -85,B 0,C 180,E1 12286.675,E2 12286.675} C_VEL
LIN {X 0,Y 267.542,Z 980.352,A -85,B 0,C 180,E1 12281.414,E2 12281.414} C_VEL
LIN {X 0,Y 270.58,Z 973.609,A -85,B 0,C 180,E1 12276.773,E2 12276.773} C_VEL
LIN {X 0,Y 274.988,Z 964.891,A -85,B 0,C 180,E1 12272.064,E2 12272.064} C_VEL
LIN {X 0,Y 280.644,Z 954.696,A -85,B 0,C 180,E1 12267.592,E2 12267.592} C_VEL
LIN {X 0,Y 287.322,Z 942.906,A -85,B 0,C 180,E1 12263.443,E2 12263.443} C_VEL
LIN {X 0,Y 295.519,Z 928.71,A -85,B 0,C 180,E1 12259.365,E2 12259.365} C_VEL
LIN {X 0,Y 303.419,Z 914.732,A -85,B 0,C 180,E1 12256.07,E2 12256.07} C_VEL
LIN {X 0,Y 312.125,Z 898.671,A -85,B 0,C 180,E1 12252.959,E2 12252.959} C_VEL
LIN {X 0,Y 321.042,Z 881.42,A -85,B 0,C 180,E1 12250.196,E2 12250.196} C_VEL
LIN {X 0,Y 329.135,Z 864.317,A -85,B 0,C 180,E1 12247.951,E2 12247.951} C_VEL
LIN {X 0,Y 337.502,Z 845.299,A -85,B 0,C 180,E1 12245.867,E2 12245.867} C_VEL
LIN {X 0,Y 344.968,Z 826.19,A -85,B 0,C 180,E1 12244.156,E2 12244.156} C_VEL
LIN {X 0,Y 352.33,Z 804.996,A -85,B 0,C 180,E1 12242.602,E2 12242.602} C_VEL
LIN {X 0,Y 358.169,Z 785.389,A -85,B 0,C 180,E1 12241.44,E2 12241.44} C_VEL
LIN {X 0,Y 363.844,Z 762.664,A -85,B 0,C 180,E1 12240.37,E2 12240.37} C_VEL
LIN {X 0,Y 367.849,Z 742.557,A -85,B 0,C 180,E1 12239.638,E2 12239.638} C_VEL
LIN {X 0,Y 371.443,Z 718.157,A -85,B 0,C 180,E1 12238.985,E2 12238.985} C_VEL
LIN {X 0,Y 389.996,Z 531.522,A -85,B 0,C 180,E1 12235.129,E2 12235.129} C_VEL
LIN {X 0,Y 387.526,Z 526.399,A -85,B 0,C 180,E1 12233.11,E2 12233.11} C_VEL
LIN {X 0,Y 386.292,Z 523.798,A -85,B 0,C 180,E1 12231.816,E2 12231.816} C_VEL
LIN {X 0,Y 384.925,Z 520.655,A -85,B 0,C 180,E1 12229.827,E2 12229.827} C_VEL
LIN {X 0,Y 383.93,Z 518.567,A -85,B 0,C 180,E1 12226.138,E2 12226.138} C_VEL
LIN {X 0,Y 385.107,Z 520.938,A -85,B 0,C 180,E1 12222.317,E2 12222.317} C_VEL
LIN {X 0,Y 387.103,Z 525.499,A -85,B 0,C 180,E1 12219.751,E2 12219.751} C_VEL
LIN {X 0,Y 388.868,Z 529.455,A -85,B 0,C 180,E1 12218.146,E2 12218.146} C_VEL
LIN {X 0,Y 389.981,Z 532.651,A -85,B 0,C 180,E1 12217.231,E2 12217.231} C_VEL
LIN {X 0,Y 370.295,Z 731.277,A -85,B 0,C 180,E1 12213.119,E2 12213.119} C_VEL
LIN {X 0,Y 366.373,Z 755.275,A -85,B 0,C 180,E1 12212.477,E2 12212.477} C_VEL
LIN {X 0,Y 361.283,Z 778.723,A -85,B 0,C 180,E1 12211.657,E2 12211.657} C_VEL
LIN {X 0,Y 355.567,Z 799.948,A -85,B 0,C 180,E1 12210.665,E2 12210.665} C_VEL
LIN {X 0,Y 348.261,Z 823.003,A -85,B 0,C 180,E1 12209.291,E2 12209.291} C_VEL
LIN {X 0,Y 341.05,Z 842.951,A -85,B 0,C 180,E1 12207.802,E2 12207.802} C_VEL
LIN {X 0,Y 332.671,Z 863.551,A -85,B 0,C 180,E1 12205.903,E2 12205.903} C_VEL
LIN {X 0,Y 324.301,Z 882.522,A -85,B 0,C 180,E1 12203.775,E2 12203.775} C_VEL
LIN {X 0,Y 315.713,Z 900.351,A -85,B 0,C 180,E1 12201.327,E2 12201.327} C_VEL
LIN {X 0,Y 306.817,Z 917.988,A -85,B 0,C 180,E1 12198.415,E2 12198.415} C_VEL
LIN {X 0,Y 298.49,Z 933.712,A -85,B 0,C 180,E1 12195.252,E2 12195.252} C_VEL
LIN {X 0,Y 290.116,Z 949.338,A -85,B 0,C 180,E1 12191.437,E2 12191.437} C_VEL
LIN {X 0,Y 282.951,Z 962.854,A -85,B 0,C 180,E1 12187.436,E2 12187.436} C_VEL
LIN {X 0,Y 276.763,Z 974.846,A -85,B 0,C 180,E1 12183.057,E2 12183.057} C_VEL
LIN {X 0,Y 271.749,Z 985.476,A -85,B 0,C 180,E1 12178.342,E2 12178.342} C_VEL
LIN {X 0,Y 268.262,Z 993.814,A -85,B 0,C 180,E1 12173.743,E2 12173.743} C_VEL
LIN {X 0,Y 265.749,Z 1001.279,A -85,B 0,C 180,E1 12168.538,E2 12168.538} C_VEL
LIN {X 0,Y 264.609,Z 1006.019,A -85,B 0,C 180,E1 12164.224,E2 12164.224} C_VEL
LIN {X 0,Y 264.066,Z 1009.891,A -85,B 0,C 180,E1 12159.377,E2 12159.377} C_VEL
LIN {X 0,Y 263.972,Z 1011.904,A -85,B 0,C 180,E1 12155.222,E2 12155.222} C_VEL
LIN {X 0,Y 263.992,Z 1012.782,A -85,B 0,C 180,E1 12151.309,E2 12151.309} C_VEL
LIN {X 0,Y 263.967,Z 1012.593,A -85,B 0,C 180,E1 12146.967,E2 12146.967} C_VEL
LIN {X 0,Y 263.979,Z 1010.966,A -85,B 0,C 180,E1 12142.608,E2 12142.608} C_VEL
LIN {X 0,Y 264.214,Z 1008.367,A -85,B 0,C 180,E1 12138.554,E2 12138.554} C_VEL
LIN {X 0,Y 265.039,Z 1003.949,A -85,B 0,C 180,E1 12133.797,E2 12133.797} C_VEL
LIN {X 0,Y 266.704,Z 997.989,A -85,B 0,C 180,E1 12129.144,E2 12129.144} C_VEL
LIN {X 0,Y 269.579,Z 990.112,A -85,B 0,C 180,E1 12124.29,E2 12124.29} C_VEL
LIN {X 0,Y 273.345,Z 981.241,A -85,B 0,C 180,E1 12119.934,E2 12119.934} C_VEL
LIN {X 0,Y 278.979,Z 969.261,A -85,B 0,C 180,E1 12115.157,E2 12115.157} C_VEL
LIN {X 0,Y 285.211,Z 956.816,A -85,B 0,C 180,E1 12111.1,E2 12111.1} C_VEL
LIN {X 0,Y 292.258,Z 942.727,A -85,B 0,C 180,E1 12107.352,E2 12107.352} C_VEL
LIN {X 0,Y 299.956,Z 927.368,A -85,B 0,C 180,E1 12103.956,E2 12103.956} C_VEL
LIN {X 0,Y 307.64,Z 911.334,A -85,B 0,C 180,E1 12101.034,E2 12101.034} C_VEL
LIN {X 0,Y 316.171,Z 892.614,A -85,B 0,C 180,E1 12098.212,E2 12098.212} C_VEL
LIN {X 0,Y 324.066,Z 874.074,A -85,B 0,C 180,E1 12095.911,E2 12095.911} C_VEL
LIN {X 0,Y 331.459,Z 854.869,A -85,B 0,C 180,E1 12093.961,E2 12093.961} C_VEL
LIN {X 0,Y 338.639,Z 834.423,A -85,B 0,C 180,E1 12092.243,E2 12092.243} C_VEL
LIN {X 0,Y 344.777,Z 814.156,A -85,B 0,C 180,E1 12090.876,E2 12090.876} C_VEL
LIN {X 0,Y 350.622,Z 792.1,A -85,B 0,C 180,E1 12089.674,E2 12089.674} C_VEL
LIN {X 0,Y 355.26,Z 770.593,A -85,B 0,C 180,E1 12088.77,E2 12088.77} C_VEL
LIN {X 0,Y 359.447,Z 745.924,A -85,B 0,C 180,E1 12087.997,E2 12087.997} C_VEL
LIN {X 0,Y 361.98,Z 723.087,A -85,B 0,C 180,E1 12087.451,E2 12087.451} C_VEL
LIN {X 0,Y 376.963,Z 528.512,A -85,B 0,C 180,E1 12083.527,E2 12083.527} C_VEL
LIN {X 0,Y 369.379,Z 515.765,A -85,B 0,C 180,E1 12080.561,E2 12080.561} C_VEL
LIN {X 0,Y 362.384,Z 504.964,A -85,B 0,C 180,E1 12077.502,E2 12077.502} C_VEL
LIN {X 0,Y 356.532,Z 497.094,A -85,B 0,C 180,E1 12074.66,E2 12074.66} C_VEL
LIN {X 0,Y 353.13,Z 492.589,A -85,B 0,C 180,E1 12072.841,E2 12072.841} C_VEL
LIN {X 0,Y 350.432,Z 488.992,A -85,B 0,C 180,E1 12071.27,E2 12071.27} C_VEL
LIN {X 0,Y 346.459,Z 483.802,A -85,B 0,C 180,E1 12068.714,E2 12068.714} C_VEL
LIN {X 0,Y 342.916,Z 479.2,A -85,B 0,C 180,E1 12066.109,E2 12066.109} C_VEL
LIN {X 0,Y 338.955,Z 474.566,A -85,B 0,C 180,E1 12062.705,E2 12062.705} C_VEL
LIN {X 0,Y 338.029,Z 472.871,A -85,B 0,C 180,E1 12061.694,E2 12061.694} C_VEL
LIN {X 0,Y 334.594,Z 469.547,A -85,B 0,C 180,E1 12057.773,E2 12057.773} C_VEL
LIN {X 0,Y 333.383,Z 466.865,A -85,B 0,C 180,E1 12055.699,E2 12055.699} C_VEL
LIN {X 0,Y 330.463,Z 464.879,A -85,B 0,C 180,E1 12048.303,E2 12048.303} C_VEL
LIN {X 0,Y 330.382,Z 464.853,A -85,B 0,C 180,E1 12043.472,E2 12043.472} C_VEL
LIN {X 0,Y 332.707,Z 466.551,A -85,B 0,C 180,E1 12036.628,E2 12036.628} C_VEL
LIN {X 0,Y 333.594,Z 467.189,A -85,B 0,C 180,E1 12035.189,E2 12035.189} C_VEL
LIN {X 0,Y 335.624,Z 470.875,A -85,B 0,C 180,E1 12032.113,E2 12032.113} C_VEL
LIN {X 0,Y 338.302,Z 473.262,A -85,B 0,C 180,E1 12029.248,E2 12029.248} C_VEL
LIN {X 0,Y 341.247,Z 477.501,A -85,B 0,C 180,E1 12026.474,E2 12026.474} C_VEL
LIN {X 0,Y 343.052,Z 479.37,A -85,B 0,C 180,E1 12025.059,E2 12025.059} C_VEL
LIN {X 0,Y 346.581,Z 483.893,A -85,B 0,C 180,E1 12022.489,E2 12022.489} C_VEL
LIN {X 0,Y 352.074,Z 491.095,A -85,B 0,C 180,E1 12019.052,E2 12019.052} C_VEL
LIN {X 0,Y 356.323,Z 496.805,A -85,B 0,C 180,E1 12016.734,E2 12016.734} C_VEL
LIN {X 0,Y 362.417,Z 505.022,A -85,B 0,C 180,E1 12013.782,E2 12013.782} C_VEL
LIN {X 0,Y 369.794,Z 515.649,A -85,B 0,C 180,E1 12010.624,E2 12010.624} C_VEL
LIN {X 0,Y 376.603,Z 526.02,A -85,B 0,C 180,E1 12008.016,E2 12008.016} C_VEL
LIN {X 0,Y 361.666,Z 717.371,A -85,B 0,C 180,E1 12004.144,E2 12004.144} C_VEL
LIN {X 0,Y 358.432,Z 741.451,A -85,B 0,C 180,E1 12003.482,E2 12003.482} C_VEL
LIN {X 0,Y 354.414,Z 763.824,A -85,B 0,C 180,E1 12002.645,E2 12002.645} C_VEL
LIN {X 0,Y 349.372,Z 785.549,A -85,B 0,C 180,E1 12001.575,E2 12001.575} C_VEL
LIN {X 0,Y 343.436,Z 807.294,A -85,B 0,C 180,E1 12000.235,E2 12000.235} C_VEL
LIN {X 0,Y 337.054,Z 827.177,A -85,B 0,C 180,E1 11998.715,E2 11998.715} C_VEL
LIN {X 0,Y 329.233,Z 848.684,A -85,B 0,C 180,E1 11996.702,E2 11996.702} C_VEL
LIN {X 0,Y 321.793,Z 867.11,A -85,B 0,C 180,E1 11994.598,E2 11994.598} C_VEL
LIN {X 0,Y 313.741,Z 885.217,A -85,B 0,C 180,E1 11992.082,E2 11992.082} C_VEL
LIN {X 0,Y 305.81,Z 902.054,A -85,B 0,C 180,E1 11989.276,E2 11989.276} C_VEL
LIN {X 0,Y 298.07,Z 917.41,A -85,B 0,C 180,E1 11986.159,E2 11986.159} C_VEL
LIN {X 0,Y 290.378,Z 932.246,A -85,B 0,C 180,E1 11982.522,E2 11982.522} C_VEL
LIN {X 0,Y 283.998,Z 944.413,A -85,B 0,C 180,E1 11978.905,E2 11978.905} C_VEL
LIN {X 0,Y 277.772,Z 956.462,A -85,B 0,C 180,E1 11974.536,E2 11974.536} C_VEL
LIN {X 0,Y 272.967,Z 966.286,A -85,B 0,C 180,E1 11970.183,E2 11970.183} C_VEL
LIN {X 0,Y 269.189,Z 974.618,A -85,B 0,C 180,E1 11965.52,E2 11965.52} C_VEL
LIN {X 0,Y 266.568,Z 981.498,A -85,B 0,C 180,E1 11960.712,E2 11960.712} C_VEL
LIN {X 0,Y 265.082,Z 986.273,A -85,B 0,C 180,E1 11956.247,E2 11956.247} C_VEL
LIN {X 0,Y 264.326,Z 989.894,A -85,B 0,C 180,E1 11951.696,E2 11951.696} C_VEL
LIN {X 0,Y 264.038,Z 992.119,A -85,B 0,C 180,E1 11947.037,E2 11947.037} C_VEL
LIN {X 0,Y 263.99,Z 992.966,A -85,B 0,C 180,E1 11943.204,E2 11943.204} C_VEL
LIN {X 0,Y 264.029,Z 992.888,A -85,B 0,C 180,E1 11938.995,E2 11938.995} C_VEL
LIN {X 0,Y 264.178,Z 991.441,A -85,B 0,C 180,E1 11934.342,E2 11934.342} C_VEL
LIN {X 0,Y 264.663,Z 988.93,A -85,B 0,C 180,E1 11930.035,E2 11930.035} C_VEL
LIN {X 0,Y 265.428,Z 986.171,A -85,B 0,C 180,E1 11926.675,E2 11926.675} C_VEL
LIN {X 0,Y 264.974,Z 984.708,A -85,B 0,C 180,E1 11925.032,E2 11925.032} C_VEL
LIN {X 0,Y 260.719,Z 980.386,A -85,B 0,C 180,E1 11920.582,E2 11920.582} C_VEL
LIN {X 0,Y 260.841,Z 978.664,A -85,B 0,C 180,E1 11919.162,E2 11919.162} C_VEL
LIN {X 0,Y 264.75,Z 970.969,A -85,B 0,C 180,E1 11914.192,E2 11914.192} C_VEL
LIN {X 0,Y 269.94,Z 961.864,A -85,B 0,C 180,E1 11909.481,E2 11909.481} C_VEL
LIN {X 0,Y 276.307,Z 951.063,A -85,B 0,C 180,E1 11905.049,E2 11905.049} C_VEL
LIN {X 0,Y 284.303,Z 937.972,A -85,B 0,C 180,E1 11900.681,E2 11900.681} C_VEL
LIN {X 0,Y 292.253,Z 924.818,A -85,B 0,C 180,E1 11897.112,E2 11897.112} C_VEL
LIN {X 0,Y 301.193,Z 909.538,A -85,B 0,C 180,E1 11893.722,E2 11893.722} C_VEL
LIN {X 0,Y 310.4,Z 893.189,A -85,B 0,C 180,E1 11890.727,E2 11890.727} C_VEL
LIN {X 0,Y 319.567,Z 875.478,A -85,B 0,C 180,E1 11888.095,E2 11888.095} C_VEL
LIN {X 0,Y 328.739,Z 856.368,A -85,B 0,C 180,E1 11885.761,E2 11885.761} C_VEL
LIN {X 0,Y 336.756,Z 837.949,A -85,B 0,C 180,E1 11883.916,E2 11883.916} C_VEL
LIN {X 0,Y 345.056,Z 816.385,A -85,B 0,C 180,E1 11882.16,E2 11882.16} C_VEL
LIN {X 0,Y 352.344,Z 794.744,A -85,B 0,C 180,E1 11880.74,E2 11880.74} C_VEL
LIN {X 0,Y 358.478,Z 772.612,A -85,B 0,C 180,E1 11879.601,E2 11879.601} C_VEL
LIN {X 0,Y 363.909,Z 748.466,A -85,B 0,C 180,E1 11878.645,E2 11878.645} C_VEL
LIN {X 0,Y 367.73,Z 726.047,A -85,B 0,C 180,E1 11877.994,E2 11877.994} C_VEL
LIN {X 0,Y 372.063,Z 685.899,A -85,B 0,C 180,E1 11877.134,E2 11877.134} C_VEL
LIN {X 0,Y 387.455,Z 537.078,A -85,B 0,C 180,E1 11874.076,E2 11874.076} C_VEL
LIN {X 0,Y 385.224,Z 531.955,A -85,B 0,C 180,E1 11871.868,E2 11871.868} C_VEL
LIN {X 0,Y 383.725,Z 528.489,A -85,B 0,C 180,E1 11869.643,E2 11869.643} C_VEL
LIN {X 0,Y 382.84,Z 526.509,A -85,B 0,C 180,E1 11866.098,E2 11866.098} C_VEL
LIN {X 0,Y 383.893,Z 528.807,A -85,B 0,C 180,E1 11862.494,E2 11862.494} C_VEL
LIN {X 0,Y 385.655,Z 533.077,A -85,B 0,C 180,E1 11860.067,E2 11860.067} C_VEL
LIN {X 0,Y 387.192,Z 536.743,A -85,B 0,C 180,E1 11858.568,E2 11858.568} C_VEL
LIN {X 0,Y 387.485,Z 537.891,A -85,B 0,C 180,E1 11858.276,E2 11858.276} C_VEL
LIN {X 0,Y 367.547,Z 730.726,A -85,B 0,C 180,E1 11854.3,E2 11854.3} C_VEL
LIN {X 0,Y 363.536,Z 754.703,A -85,B 0,C 180,E1 11853.668,E2 11853.668} C_VEL
LIN {X 0,Y 358.382,Z 777.802,A -85,B 0,C 180,E1 11852.878,E2 11852.878} C_VEL
LIN {X 0,Y 352.502,Z 798.969,A -85,B 0,C 180,E1 11851.908,E2 11851.908} C_VEL
LIN {X 0,Y 345.012,Z 821.978,A -85,B 0,C 180,E1 11850.565,E2 11850.565} C_VEL
LIN {X 0,Y 337.445,Z 842.199,A -85,B 0,C 180,E1 11849.076,E2 11849.076} C_VEL
LIN {X 0,Y 329.011,Z 862.267,A -85,B 0,C 180,E1 11847.253,E2 11847.253} C_VEL
LIN {X 0,Y 319.778,Z 882.403,A -85,B 0,C 180,E1 11845.011,E2 11845.011} C_VEL
LIN {X 0,Y 310.784,Z 900.26,A -85,B 0,C 180,E1 11842.552,E2 11842.552} C_VEL
LIN {X 0,Y 301.654,Z 917.579,A -85,B 0,C 180,E1 11839.678,E2 11839.678} C_VEL
LIN {X 0,Y 292.699,Z 933.706,A -85,B 0,C 180,E1 11836.408,E2 11836.408} C_VEL
LIN {X 0,Y 283.901,Z 949.238,A -85,B 0,C 180,E1 11832.553,E2 11832.553} C_VEL
LIN {X 0,Y 276.349,Z 962.703,A -85,B 0,C 180,E1 11828.491,E2 11828.491} C_VEL
LIN {X 0,Y 269.794,Z 974.631,A -85,B 0,C 180,E1 11824.035,E2 11824.035} C_VEL
LIN {X 0,Y 264.337,Z 985.427,A -85,B 0,C 180,E1 11819.103,E2 11819.103} C_VEL
LIN {X 0,Y 260.679,Z 993.562,A -85,B 0,C 180,E1 11814.478,E2 11814.478} C_VEL
LIN {X 0,Y 257.982,Z 1000.868,A -85,B 0,C 180,E1 11809.241,E2 11809.241} C_VEL
LIN {X 0,Y 256.726,Z 1005.522,A -85,B 0,C 180,E1 11804.901,E2 11804.901} C_VEL
LIN {X 0,Y 256.085,Z 1009.477,A -85,B 0,C 180,E1 11799.899,E2 11799.899} C_VEL
LIN {X 0,Y 255.976,Z 1011.609,A -85,B 0,C 180,E1 11795.386,E2 11795.386} C_VEL
LIN {X 0,Y 255.998,Z 1012.484,A -85,B 0,C 180,E1 11791.35,E2 11791.35} C_VEL
LIN {X 0,Y 255.971,Z 1012.283,A -85,B 0,C 180,E1 11786.872,E2 11786.872} C_VEL
LIN {X 0,Y 255.991,Z 1010.643,A -85,B 0,C 180,E1 11782.376,E2 11782.376} C_VEL
LIN {X 0,Y 256.236,Z 1008.109,A -85,B 0,C 180,E1 11778.3,E2 11778.3} C_VEL
LIN {X 0,Y 257.166,Z 1003.586,A -85,B 0,C 180,E1 11773.287,E2 11773.287} C_VEL
LIN {X 0,Y 258.977,Z 997.611,A -85,B 0,C 180,E1 11768.491,E2 11768.491} C_VEL
LIN {X 0,Y 262.084,Z 989.697,A -85,B 0,C 180,E1 11763.498,E2 11763.498} C_VEL
LIN {X 0,Y 266.12,Z 980.793,A -85,B 0,C 180,E1 11759.029,E2 11759.029} C_VEL
LIN {X 0,Y 271.977,Z 969.032,A -85,B 0,C 180,E1 11754.24,E2 11754.24} C_VEL
LIN {X 0,Y 278.275,Z 957.056,A -85,B 0,C 180,E1 11750.251,E2 11750.251} C_VEL
LIN {X 0,Y 285.667,Z 942.97,A -85,B 0,C 180,E1 11746.419,E2 11746.419} C_VEL
LIN {X 0,Y 293.702,Z 927.638,A -85,B 0,C 180,E1 11742.963,E2 11742.963} C_VEL
LIN {X 0,Y 301.639,Z 911.714,A -85,B 0,C 180,E1 11740.019,E2 11740.019} C_VEL
LIN {X 0,Y 310.217,Z 893.645,A -85,B 0,C 180,E1 11737.253,E2 11737.253} C_VEL
LIN {X 0,Y 318.086,Z 875.759,A -85,B 0,C 180,E1 11735.001,E2 11735.001} C_VEL
LIN {X 0,Y 326.252,Z 855.443,A -85,B 0,C 180,E1 11732.903,E2 11732.903} C_VEL
LIN {X 0,Y 333.297,Z 836.032,A -85,B 0,C 180,E1 11731.257,E2 11731.257} C_VEL
LIN {X 0,Y 340.068,Z 814.603,A -85,B 0,C 180,E1 11729.794,E2 11729.794} C_VEL
LIN {X 0,Y 345.936,Z 793.237,A -85,B 0,C 180,E1 11728.621,E2 11728.621} C_VEL
LIN {X 0,Y 350.864,Z 771.049,A -85,B 0,C 180,E1 11727.687,E2 11727.687} C_VEL
LIN {X 0,Y 355.063,Z 747.335,A -85,B 0,C 180,E1 11726.938,E2 11726.938} C_VEL
LIN {X 0,Y 357.697,Z 724.755,A -85,B 0,C 180,E1 11726.393,E2 11726.393} C_VEL
LIN {X 0,Y 372.986,Z 533.005,A -85,B 0,C 180,E1 11722.519,E2 11722.519} C_VEL
LIN {X 0,Y 366.528,Z 522.075,A -85,B 0,C 180,E1 11719.895,E2 11719.895} C_VEL
LIN {X 0,Y 359.986,Z 511.815,A -85,B 0,C 180,E1 11716.955,E2 11716.955} C_VEL
LIN {X 0,Y 352.737,Z 501.829,A -85,B 0,C 180,E1 11713.273,E2 11713.273} C_VEL
LIN {X 0,Y 348.672,Z 496.49,A -85,B 0,C 180,E1 11710.909,E2 11710.909} C_VEL
LIN {X 0,Y 344.759,Z 491.327,A -85,B 0,C 180,E1 11708.337,E2 11708.337} C_VEL
LIN {X 0,Y 340.669,Z 486.045,A -85,B 0,C 180,E1 11705.22,E2 11705.22} C_VEL
LIN {X 0,Y 337.51,Z 482.192,A -85,B 0,C 180,E1 11702.376,E2 11702.376} C_VEL
LIN {X 0,Y 336.57,Z 480.614,A -85,B 0,C 180,E1 11701.361,E2 11701.361} C_VEL
LIN {X 0,Y 333.363,Z 477.388,A -85,B 0,C 180,E1 11697.593,E2 11697.593} C_VEL
LIN {X 0,Y 332.166,Z 474.742,A -85,B 0,C 180,E1 11695.511,E2 11695.511} C_VEL
LIN {X 0,Y 329.367,Z 472.801,A -85,B 0,C 180,E1 11688.264,E2 11688.264} C_VEL
LIN {X 0,Y 329.304,Z 472.783,A -85,B 0,C 180,E1 11683.416,E2 11683.416} C_VEL
LIN {X 0,Y 331.783,Z 474.562,A -85,B 0,C 180,E1 11676.349,E2 11676.349} C_VEL
LIN {X 0,Y 332.427,Z 475.198,A -85,B 0,C 180,E1 11675.286,E2 11675.286} C_VEL
LIN {X 0,Y 334.597,Z 478.966,A -85,B 0,C 180,E1 11672.02,E2 11672.02} C_VEL
LIN {X 0,Y 337.017,Z 481.199,A -85,B 0,C 180,E1 11669.415,E2 11669.415} C_VEL
LIN {X 0,Y 340.052,Z 485.452,A -85,B 0,C 180,E1 11666.542,E2 11666.542} C_VEL
LIN {X 0,Y 341.636,Z 487.226,A -85,B 0,C 180,E1 11665.27,E2 11665.27} C_VEL
LIN {X 0,Y 346.053,Z 493.004,A -85,B 0,C 180,E1 11662.061,E2 11662.061} C_VEL
LIN {X 0,Y 350.309,Z 498.612,A -85,B 0,C 180,E1 11659.4,E2 11659.4} C_VEL
LIN {X 0,Y 354.504,Z 504.341,A -85,B 0,C 180,E1 11657.067,E2 11657.067} C_VEL
LIN {X 0,Y 360.354,Z 512.382,A -85,B 0,C 180,E1 11654.171,E2 11654.171} C_VEL
LIN {X 0,Y 367.413,Z 522.711,A -85,B 0,C 180,E1 11651.077,E2 11651.077} C_VEL
LIN {X 0,Y 372.609,Z 530.751,A -85,B 0,C 180,E1 11649.019,E2 11649.019} C_VEL
LIN {X 0,Y 357.486,Z 718.303,A -85,B 0,C 180,E1 11645.223,E2 11645.223} C_VEL
LIN {X 0,Y 354.167,Z 742.147,A -85,B 0,C 180,E1 11644.565,E2 11644.565} C_VEL
LIN {X 0,Y 350.081,Z 764.295,A -85,B 0,C 180,E1 11643.738,E2 11643.738} C_VEL
LIN {X 0,Y 344.75,Z 786.631,A -85,B 0,C 180,E1 11642.638,E2 11642.638} C_VEL
LIN {X 0,Y 338.646,Z 808.217,A -85,B 0,C 180,E1 11641.301,E2 11641.301} C_VEL
LIN {X 0,Y 332.085,Z 828.044,A -85,B 0,C 180,E1 11639.781,E2 11639.781} C_VEL
LIN {X 0,Y 324.026,Z 849.459,A -85,B 0,C 180,E1 11637.764,E2 11637.764} C_VEL
LIN {X 0,Y 316.089,Z 868.522,A -85,B 0,C 180,E1 11635.573,E2 11635.573} C_VEL
LIN {X 0,Y 307.779,Z 886.494,A -85,B 0,C 180,E1 11633.038,E2 11633.038} C_VEL
LIN {X 0,Y 299.337,Z 903.622,A -85,B 0,C 180,E1 11630.116,E2 11630.116} C_VEL
LIN {X 0,Y 291.77,Z 918.067,A -85,B 0,C 180,E1 11627.133,E2 11627.133} C_VEL
LIN {X 0,Y 283.381,Z 933.552,A -85,B 0,C 180,E1 11623.251,E2 11623.251} C_VEL
LIN {X 0,Y 276.77,Z 945.645,A -85,B 0,C 180,E1 11619.559,E2 11619.559} C_VEL
LIN {X 0,Y 270.557,Z 957.025,A -85,B 0,C 180,E1 11615.294,E2 11615.294} C_VEL
LIN {X 0,Y 265.523,Z 966.787,A -85,B 0,C 180,E1 11610.856,E2 11610.856} C_VEL
LIN {X 0,Y 261.512,Z 975.122,A -85,B 0,C 180,E1 11606.047,E2 11606.047} C_VEL
LIN {X 0,Y 258.734,Z 981.942,A -85,B 0,C 180,E1 11601.101,E2 11601.101} C_VEL
LIN {X 0,Y 257.136,Z 986.747,A -85,B 0,C 180,E1 11596.44,E2 11596.44} C_VEL
LIN {X 0,Y 256.319,Z 990.433,A -85,B 0,C 180,E1 11591.574,E2 11591.574} C_VEL
LIN {X 0,Y 256.043,Z 992.458,A -85,B 0,C 180,E1 11587.008,E2 11587.008} C_VEL
LIN {X 0,Y 255.995,Z 993.282,A -85,B 0,C 180,E1 11583.053,E2 11583.053} C_VEL
LIN {X 0,Y 256.036,Z 993.18,A -85,B 0,C 180,E1 11578.702,E2 11578.702} C_VEL
LIN {X 0,Y 256.218,Z 991.668,A -85,B 0,C 180,E1 11573.882,E2 11573.882} C_VEL
LIN {X 0,Y 256.79,Z 989.103,A -85,B 0,C 180,E1 11569.401,E2 11569.401} C_VEL
LIN {X 0,Y 258.274,Z 984.598,A -85,B 0,C 180,E1 11564.175,E2 11564.175} C_VEL
LIN {X 0,Y 260.603,Z 979.142,A -85,B 0,C 180,E1 11559.532,E2 11559.532} C_VEL
LIN {X 0,Y 260.841,Z 978.664,A -85,B 0,C 180,E1 11559.162,E2 11559.162} C_VEL
LIN {X 0,Y 260.993,Z 976.593,A -85,B 0,C 180,E1 11557.52,E2 11557.52} C_VEL
LIN {X 0,Y 258.527,Z 970.733,A -85,B 0,C 180,E1 11553.041,E2 11553.041} C_VEL
LIN {X 0,Y 259.234,Z 968.524,A -85,B 0,C 180,E1 11551.656,E2 11551.656} C_VEL
LIN {X 0,Y 265.233,Z 958.708,A -85,B 0,C 180,E1 11546.897,E2 11546.897} C_VEL
LIN {X 0,Y 272.577,Z 947.323,A -85,B 0,C 180,E1 11542.414,E2 11542.414} C_VEL
LIN {X 0,Y 280.5,Z 934.965,A -85,B 0,C 180,E1 11538.497,E2 11538.497} C_VEL
LIN {X 0,Y 290.134,Z 919.683,A -85,B 0,C 180,E1 11534.571,E2 11534.571} C_VEL
LIN {X 0,Y 298.994,Z 905.13,A -85,B 0,C 180,E1 11531.514,E2 11531.514} C_VEL
LIN {X 0,Y 308.487,Z 888.469,A -85,B 0,C 180,E1 11528.654,E2 11528.654} C_VEL
LIN {X 0,Y 318.027,Z 870.64,A -85,B 0,C 180,E1 11526.137,E2 11526.137} C_VEL
LIN {X 0,Y 326.869,Z 852.351,A -85,B 0,C 180,E1 11524.035,E2 11524.035} C_VEL
LIN {X 0,Y 335.712,Z 832.207,A -85,B 0,C 180,E1 11522.134,E2 11522.134} C_VEL
LIN {X 0,Y 343.084,Z 813.109,A -85,B 0,C 180,E1 11520.669,E2 11520.669} C_VEL
LIN {X 0,Y 350.455,Z 791.168,A -85,B 0,C 180,E1 11519.306,E2 11519.306} C_VEL
LIN {X 0,Y 356.121,Z 771.084,A -85,B 0,C 180,E1 11518.311,E2 11518.311} C_VEL
LIN {X 0,Y 361.391,Z 748.008,A -85,B 0,C 180,E1 11517.424,E2 11517.424} C_VEL
LIN {X 0,Y 365.422,Z 724.957,A -85,B 0,C 180,E1 11516.772,E2 11516.772} C_VEL
LIN {X 0,Y 373.321,Z 651.475,A -85,B 0,C 180,E1 11515.24,E2 11515.24} C_VEL
LIN {X 0,Y 385.152,Z 542.728,A -85,B 0,C 180,E1 11513.034,E2 11513.034} C_VEL
LIN {X 0,Y 383.628,Z 539.201,A -85,B 0,C 180,E1 11511.306,E2 11511.306} C_VEL
LIN {X 0,Y 382.495,Z 536.283,A -85,B 0,C 180,E1 11509.395,E2 11509.395} C_VEL
LIN {X 0,Y 381.75,Z 534.452,A -85,B 0,C 180,E1 11506.057,E2 11506.057} C_VEL
LIN {X 0,Y 382.718,Z 536.814,A -85,B 0,C 180,E1 11502.595,E2 11502.595} C_VEL
LIN {X 0,Y 384.284,Z 540.827,A -85,B 0,C 180,E1 11500.31,E2 11500.31} C_VEL
LIN {X 0,Y 385.184,Z 543.209,A -85,B 0,C 180,E1 11499.335,E2 11499.335} C_VEL
LIN {X 0,Y 364.96,Z 730.986,A -85,B 0,C 180,E1 11495.487,E2 11495.487} C_VEL
LIN {X 0,Y 360.8,Z 754.822,A -85,B 0,C 180,E1 11494.862,E2 11494.862} C_VEL
LIN {X 0,Y 355.275,Z 778.518,A -85,B 0,C 180,E1 11494.057,E2 11494.057} C_VEL
LIN {X 0,Y 348.881,Z 800.709,A -85,B 0,C 180,E1 11493.043,E2 11493.043} C_VEL
LIN {X 0,Y 341.192,Z 823.142,A -85,B 0,C 180,E1 11491.723,E2 11491.723} C_VEL
LIN {X 0,Y 332.817,Z 844.631,A -85,B 0,C 180,E1 11490.13,E2 11490.13} C_VEL
LIN {X 0,Y 323.9,Z 864.657,A -85,B 0,C 180,E1 11488.267,E2 11488.267} C_VEL
LIN {X 0,Y 314.239,Z 884.598,A -85,B 0,C 180,E1 11485.989,E2 11485.989} C_VEL
LIN {X 0,Y 304.853,Z 902.469,A -85,B 0,C 180,E1 11483.477,E2 11483.477} C_VEL
LIN {X 0,Y 295.291,Z 919.546,A -85,B 0,C 180,E1 11480.541,E2 11480.541} C_VEL
LIN {X 0,Y 286.444,Z 934.771,A -85,B 0,C 180,E1 11477.378,E2 11477.378} C_VEL
LIN {X 0,Y 277.59,Z 949.536,A -85,B 0,C 180,E1 11473.617,E2 11473.617} C_VEL
LIN {X 0,Y 269.484,Z 963.174,A -85,B 0,C 180,E1 11469.386,E2 11469.386} C_VEL
LIN {X 0,Y 262.895,Z 974.452,A -85,B 0,C 180,E1 11465.057,E2 11465.057} C_VEL
LIN {X 0,Y 257.162,Z 985.024,A -85,B 0,C 180,E1 11460.11,E2 11460.11} C_VEL
LIN {X 0,Y 253.109,Z 993.371,A -85,B 0,C 180,E1 11455.23,E2 11455.23} C_VEL
LIN {X 0,Y 250.204,Z 1000.604,A -85,B 0,C 180,E1 11449.864,E2 11449.864} C_VEL
